C01821=1188.862,-40.963,-42.366,179.700,5.675,149.093
C01822=1188.867,-41.212,-42.354,179.698,5.675,149.094
C01823=1188.872,-41.462,-42.342,179.695,5.674,149.094
C01824=1188.878,-41.712,-42.330,179.693,5.675,149.095
C01825=1188.883,-41.961,-42.318,179.691,5.674,149.095
C01826=1188.888,-42.211,-42.306,179.688,5.673,149.096
C01827=1188.893,-42.460,-42.294,179.686,5.673,149.097
C01828=1188.898,-42.710,-42.282,179.683,5.673,149.097
C01829=1188.903,-42.960,-42.270,179.681,5.673,149.098
C01830=1188.909,-43.209,-42.258,179.679,5.672,149.099
C01831=1188.914,-43.459,-42.246,179.676,5.672,149.099
C01832=1188.919,-43.709,-42.234,179.674,5.672,149.100
C01833=1188.924,-43.959,-42.223,179.672,5.671,149.101
C01834=1188.929,-44.208,-42.210,179.669,5.671,149.101
C01835=1188.935,-44.458,-42.198,179.667,5.671,149.102
C01836=1188.939,-44.708,-42.187,179.664,5.671,149.103
C01837=1188.944,-44.957,-42.174,179.662,5.670,149.103
C01838=1188.950,-45.207,-42.162,179.659,5.669,149.104
C01839=1188.955,-45.457,-42.150,179.657,5.670,149.105
C01840=1188.961,-45.706,-42.139,179.655,5.669,149.105
C01841=1188.966,-45.955,-42.127,179.653,5.668,149.106
C01842=1188.971,-46.205,-42.115,179.650,5.668,149.106
C01843=1188.977,-46.455,-42.103,179.648,5.668,149.107
C01844=1188.981,-46.705,-42.092,179.646,5.668,149.108
C01845=1188.986,-46.954,-42.079,179.643,5.667,149.108
C01846=1188.992,-47.204,-42.067,179.640,5.667,149.109
C01847=1188.997,-47.454,-42.056,179.638,5.667,149.110
C01848=1189.002,-47.704,-42.044,179.636,5.666,149.110
C01849=1189.007,-47.954,-42.032,179.633,5.666,149.111
C01850=1189.012,-48.203,-42.020,179.631,5.666,149.112
C01851=1189.017,-48.452,-42.008,179.629,5.666,149.112
C01852=1189.023,-48.702,-41.996,179.626,5.665,149.113
C01853=1189.027,-48.952,-41.985,179.624,5.664,149.113
C01854=1189.033,-49.222,-41.973,179.621,5.664,149.114
C01855=1189.039,-49.492,-41.960,179.619,5.664,149.115
C01856=1189.045,-49.762,-41.948,179.616,5.664,149.116
C01857=1189.051,-50.033,-41.934,179.614,5.664,149.116
C01858=1189.055,-50.283,-41.923,179.611,5.663,149.117
C01859=1189.061,-50.533,-41.911,179.609,5.662,149.117
C01860=1189.065,-50.782,-41.899,179.607,5.663,149.118
C01861=1189.071,-51.031,-41.887,179.604,5.662,149.119
C01862=1189.077,-51.281,-41.876,179.601,5.662,149.120
C01863=1189.081,-51.530,-41.864,179.600,5.662,149.120
C01864=1189.087,-51.780,-41.852,179.597,5.661,149.121
C01865=1189.092,-52.030,-41.841,179.595,5.661,149.121
C01866=1189.097,-52.280,-41.829,179.592,5.661,149.122
C01867=1189.102,-52.530,-41.817,179.590,5.660,149.123
C01868=1189.107,-52.779,-41.806,179.588,5.660,149.123
C01869=1189.113,-53.029,-41.795,179.585,5.660,149.124
C01870=1189.118,-53.278,-41.783,179.583,5.660,149.125
C01871=1189.123,-53.528,-41.771,179.581,5.659,149.125
C01872=1189.128,-53.778,-41.760,179.578,5.659,149.126
C01873=1189.133,-54.028,-41.748,179.576,5.659,149.127
C01874=1189.138,-54.277,-41.737,179.573,5.659,149.127
C01875=1189.144,-54.527,-41.725,179.571,5.658,149.128
C01876=1189.150,-54.777,-41.713,179.568,5.657,149.128
C01877=1189.154,-55.026,-41.702,179.566,5.658,149.129
C01878=1189.160,-55.276,-41.690,179.564,5.657,149.130
C01879=1189.164,-55.526,-41.679,179.561,5.656,149.130
C01880=1189.170,-55.776,-41.667,179.559,5.657,149.131
C01881=1189.174,-56.025,-41.656,179.557,5.656,149.132
C01882=1189.181,-56.275,-41.644,179.555,5.656,149.132
C01883=1189.185,-56.524,-41.633,179.552,5.656,149.133
C01884=1189.191,-56.774,-41.621,179.550,5.655,149.134
C01885=1189.195,-57.024,-41.610,179.547,5.655,149.134
C01886=1189.201,-57.274,-41.598,179.546,5.655,149.135
C01887=1189.206,-57.523,-41.587,179.543,5.655,149.136
C01888=1189.211,-57.772,-41.576,179.540,5.654,149.136
C01889=1189.216,-58.023,-41.565,179.538,5.654,149.137
C01890=1189.221,-58.272,-41.553,179.536,5.654,149.137
C01891=1189.227,-58.522,-41.542,179.533,5.653,149.138
C01892=1189.232,-58.771,-41.530,179.531,5.653,149.139
C01893=1189.237,-59.021,-41.519,179.529,5.653,149.139
C01894=1189.242,-59.271,-41.507,179.526,5.652,149.140
C01895=1189.247,-59.521,-41.495,179.524,5.652,149.141
C01896=1189.253,-59.770,-41.484,179.522,5.652,149.141
C01897=1189.258,-60.020,-41.474,179.519,5.652,149.142
C01898=1189.263,-60.270,-41.462,179.517,5.651,149.143
C01899=1189.268,-60.519,-41.451,179.515,5.651,149.143
C01900=1189.274,-60.769,-41.439,179.512,5.651,149.144
C01901=1189.279,-61.018,-41.428,179.510,5.650,149.145
C01902=1189.284,-61.269,-41.417,179.508,5.651,149.145
C01903=1189.289,-61.519,-41.405,179.505,5.650,149.146
C01904=1189.294,-61.767,-41.395,179.503,5.649,149.146
C01905=1189.300,-62.017,-41.383,179.501,5.650,149.147
C01906=1189.304,-62.267,-41.371,179.498,5.649,149.148
C01907=1189.310,-62.517,-41.361,179.495,5.649,149.149
C01908=1189.315,-62.766,-41.349,179.494,5.649,149.149
C01909=1189.320,-63.016,-41.338,179.491,5.648,149.150
C01910=1189.326,-63.266,-41.326,179.489,5.648,149.150
C01911=1189.331,-63.516,-41.316,179.487,5.648,149.151
C01912=1189.336,-63.765,-41.305,179.484,5.648,149.152
C01913=1189.341,-64.015,-41.293,179.482,5.647,149.152
C01914=1189.347,-64.265,-41.283,179.480,5.648,149.153
C01915=1189.352,-64.514,-41.271,179.477,5.647,149.153
C01916=1189.357,-64.764,-41.259,179.475,5.646,149.154
C01917=1189.362,-65.013,-41.248,179.473,5.647,149.155
C01918=1189.367,-65.263,-41.238,179.470,5.646,149.155
C01919=1189.373,-65.513,-41.226,179.468,5.645,149.156
C01920=1189.378,-65.762,-41.215,179.466,5.646,149.157
C01921=1189.383,-66.013,-41.204,179.463,5.645,149.157
C01922=1189.388,-66.262,-41.193,179.461,5.645,149.158
C01923=1189.394,-66.511,-41.182,179.459,5.645,149.159
C01924=1189.399,-66.762,-41.171,179.456,5.644,149.159
C01925=1189.403,-67.011,-41.160,179.454,5.644,149.160
C01926=1189.410,-67.261,-41.149,179.452,5.644,149.161
C01927=1189.414,-67.511,-41.138,179.449,5.644,149.161
C01928=1189.419,-67.760,-41.126,179.446,5.643,149.162
C01929=1189.425,-68.010,-41.116,179.445,5.643,149.162
C01930=1189.430,-68.260,-41.104,179.442,5.643,149.163
C01931=1189.435,-68.510,-41.094,179.440,5.643,149.164
C01932=1189.440,-68.759,-41.083,179.438,5.642,149.164
C01933=1189.445,-69.009,-41.072,179.435,5.642,149.165
C01934=1189.451,-69.259,-41.060,179.433,5.642,149.166
C01935=1189.456,-69.508,-41.049,179.430,5.642,149.166
C01936=1189.461,-69.758,-41.039,179.428,5.641,149.167
C01937=1189.466,-70.007,-41.028,179.426,5.641,149.168
C01938=1189.472,-70.258,-41.017,179.424,5.641,149.168
C01939=1189.477,-70.507,-41.005,179.421,5.640,149.169
C01940=1189.482,-70.757,-40.995,179.419,5.641,149.170
C01941=1189.487,-71.007,-40.984,179.417,5.640,149.170
C01942=1189.493,-71.256,-40.974,179.414,5.639,149.171
C01943=1189.498,-71.506,-40.962,179.412,5.640,149.171
C01944=1189.503,-71.756,-40.951,179.410,5.639,149.172
C01945=1189.509,-72.005,-40.940,179.408,5.640,149.173
C01946=1189.514,-72.256,-40.930,179.405,5.639,149.173
C01947=1189.519,-72.504,-40.919,179.403,5.638,149.174
C01948=1189.525,-72.755,-40.908,179.401,5.639,149.175
C01949=1189.530,-73.004,-40.897,179.398,5.638,149.175
C01950=1189.535,-73.254,-40.886,179.396,5.638,149.176
C01951=1189.540,-73.504,-40.875,179.394,5.638,149.177
C01952=1189.545,-73.753,-40.865,179.392,5.637,149.177
C01953=1189.550,-74.003,-40.853,179.389,5.638,149.178
C01954=1189.555,-74.253,-40.843,179.387,5.637,149.179
C01955=1189.561,-74.503,-40.832,179.384,5.637,149.179
C01956=1189.566,-74.752,-40.821,179.383,5.637,149.180
C01957=1189.571,-75.002,-40.811,179.380,5.636,149.180
C01958=1189.578,-75.273,-40.799,179.377,5.636,149.181
C01959=1189.583,-75.543,-40.787,179.374,5.635,149.182
C01960=1189.588,-75.815,-40.775,179.372,5.636,149.183
C01961=1189.595,-76.085,-40.764,179.370,5.635,149.183
C01962=1189.600,-76.335,-40.753,179.368,5.635,149.184
C01963=1189.605,-76.584,-40.742,179.365,5.635,149.184
C01964=1189.610,-76.834,-40.732,179.363,5.635,149.185
C01965=1189.616,-77.084,-40.721,179.361,5.635,149.186
C01966=1189.620,-77.334,-40.710,179.359,5.634,149.186
C01967=1189.626,-77.583,-40.700,179.356,5.634,149.187
C01968=1189.631,-77.833,-40.689,179.354,5.634,149.188
C01969=1189.636,-78.082,-40.678,179.352,5.633,149.188
C01970=1189.641,-78.333,-40.668,179.349,5.633,149.189
C01971=1189.647,-78.582,-40.658,179.347,5.633,149.190
C01972=1189.652,-78.832,-40.647,179.345,5.632,149.190
C01973=1189.657,-79.081,-40.636,179.343,5.633,149.191
C01974=1189.662,-79.332,-40.625,179.340,5.632,149.192
C01975=1189.668,-79.581,-40.615,179.338,5.632,149.192
C01976=1189.673,-79.831,-40.603,179.336,5.632,149.193
C01977=1189.679,-80.081,-40.593,179.333,5.632,149.193
C01978=1189.684,-80.331,-40.583,179.331,5.632,149.194
C01979=1189.689,-80.580,-40.572,179.329,5.631,149.195
C01980=1189.694,-80.830,-40.561,179.326,5.631,149.195
C01981=1189.700,-81.080,-40.551,179.324,5.631,149.196
C01982=1189.705,-81.330,-40.540,179.322,5.630,149.197
C01983=1189.710,-81.579,-40.530,179.320,5.631,149.197
C01984=1189.715,-81.830,-40.519,179.317,5.630,149.198
C01985=1189.720,-82.079,-40.509,179.315,5.630,149.198
C01986=1189.725,-82.329,-40.498,179.313,5.630,149.199
C01987=1189.730,-82.578,-40.488,179.311,5.629,149.200
C01988=1189.736,-82.828,-40.478,179.308,5.630,149.200
C01989=1189.741,-83.078,-40.468,179.306,5.629,149.201
C01990=1189.746,-83.327,-40.457,179.304,5.628,149.202
C01991=1189.751,-83.577,-40.446,179.302,5.629,149.202
C01992=1189.757,-83.826,-40.436,179.299,5.628,149.203
C01993=1189.762,-84.077,-40.425,179.297,5.628,149.203
C01994=1189.767,-84.326,-40.415,179.295,5.628,149.204
C01995=1189.773,-84.576,-40.405,179.292,5.627,149.205
C01996=1189.778,-84.825,-40.394,179.290,5.627,149.205
C01997=1189.783,-85.075,-40.383,179.288,5.627,149.206
C01998=1189.788,-85.325,-40.373,179.286,5.627,149.207
C01999=1189.794,-85.575,-40.363,179.283,5.627,149.207
C02000=1189.799,-85.825,-40.352,179.281,5.626,149.208
C02001=1189.804,-86.074,-40.342,179.279,5.627,149.209
C02002=1189.809,-86.324,-40.332,179.276,5.626,149.209
C02003=1189.814,-86.574,-40.322,179.274,5.626,149.210
C02004=1189.820,-86.824,-40.311,179.272,5.626,149.211
C02005=1189.825,-87.073,-40.301,179.270,5.626,149.211
C02006=1189.830,-87.323,-40.291,179.267,5.625,149.212
C02007=1189.836,-87.572,-40.280,179.265,5.625,149.212
C02008=1189.841,-87.823,-40.269,179.263,5.625,149.213
C02009=1189.846,-88.072,-40.260,179.260,5.625,149.214
C02010=1189.851,-88.321,-40.249,179.258,5.625,149.214
C02011=1189.856,-88.572,-40.239,179.256,5.624,149.215
C02012=1189.862,-88.821,-40.229,179.253,5.624,149.216
C02013=1189.867,-89.071,-40.218,179.251,5.624,149.216
C02014=1189.872,-89.321,-40.208,179.249,5.623,149.217
C02015=1189.877,-89.570,-40.198,179.247,5.624,149.217
C02016=1189.883,-89.820,-40.188,179.244,5.623,149.218
C02017=1189.888,-90.070,-40.177,179.243,5.623,149.219
C02018=1189.893,-90.319,-40.167,179.240,5.623,149.219
C02019=1189.898,-90.570,-40.157,179.238,5.623,149.220
C02020=1189.903,-90.819,-40.147,179.236,5.622,149.221
C02021=1189.909,-91.068,-40.137,179.233,5.622,149.221
C02022=1189.914,-91.319,-40.126,179.232,5.622,149.222
C02023=1189.920,-91.568,-40.116,179.229,5.622,149.222
C02024=1189.925,-91.818,-40.106,179.227,5.622,149.223
C02025=1189.930,-92.068,-40.097,179.225,5.621,149.224
C02026=1189.935,-92.318,-40.086,179.222,5.621,149.224
C02027=1189.941,-92.567,-40.076,179.220,5.621,149.225
C02028=1189.946,-92.817,-40.066,179.218,5.620,149.226
C02029=1189.951,-93.067,-40.055,179.216,5.621,149.226
C02030=1189.956,-93.316,-40.046,179.213,5.620,149.227
C02031=1189.962,-93.566,-40.035,179.211,5.620,149.227
C02032=1189.967,-93.816,-40.025,179.209,5.620,149.228
C02033=1189.973,-94.066,-40.015,179.207,5.620,149.229
C02034=1189.977,-94.315,-40.005,179.204,5.620,149.229
C02035=1189.983,-94.565,-39.996,179.202,5.619,149.230
C02036=1189.988,-94.815,-39.985,179.200,5.619,149.231
C02037=1189.993,-95.065,-39.975,179.198,5.619,149.231
C02038=1189.999,-95.314,-39.965,179.195,5.619,149.232
C02039=1190.004,-95.564,-39.955,179.193,5.618,149.232
C02040=1190.009,-95.814,-39.944,179.191,5.619,149.233
C02041=1190.015,-96.064,-39.936,179.188,5.618,149.234
C02042=1190.020,-96.313,-39.925,179.187,5.618,149.234
C02043=1190.025,-96.564,-39.915,179.184,5.618,149.235
C02044=1190.030,-96.813,-39.905,179.182,5.618,149.236
C02045=1190.036,-97.062,-39.895,179.180,5.618,149.236
C02046=1190.041,-97.313,-39.885,179.177,5.617,149.237
C02047=1190.046,-97.563,-39.875,179.176,5.617,149.237
C02048=1190.051,-97.812,-39.865,179.173,5.617,149.238
C02049=1190.057,-98.062,-39.855,179.171,5.617,149.239
C02050=1190.062,-98.311,-39.845,179.169,5.616,149.239
C02051=1190.068,-98.561,-39.836,179.167,5.617,149.240
C02052=1190.073,-98.811,-39.825,179.164,5.616,149.241
C02053=1190.078,-99.060,-39.816,179.162,5.616,149.241
C02054=1190.083,-99.310,-39.806,179.160,5.616,149.242
C02055=1190.089,-99.560,-39.796,179.157,5.615,149.243
C02056=1190.093,-99.810,-39.786,179.155,5.616,149.243
C02057=1190.099,-100.060,-39.776,179.153,5.615,149.244
C02058=1190.105,-100.310,-39.766,179.151,5.615,149.244
C02059=1190.110,-100.559,-39.757,179.148,5.615,149.245
C02060=1190.115,-100.809,-39.747,179.147,5.615,149.246
C02061=1190.120,-101.059,-39.737,179.144,5.614,149.246
C02062=1190.126,-101.330,-39.726,179.142,5.615,149.247
C02063=1190.132,-101.602,-39.716,179.139,5.614,149.248
C02064=1190.137,-101.873,-39.705,179.137,5.614,149.248
C02065=1190.143,-102.146,-39.694,179.135,5.614,149.249
C02066=1190.148,-102.395,-39.684,179.132,5.614,149.250
C02067=1190.154,-102.644,-39.674,179.130,5.613,149.250
C02068=1190.159,-102.894,-39.665,179.128,5.613,149.251
C02069=1190.165,-103.144,-39.655,179.126,5.613,149.252
C02070=1190.169,-103.394,-39.645,179.124,5.613,149.252
C02071=1190.175,-103.644,-39.636,179.121,5.612,149.253
C02072=1190.180,-103.893,-39.625,179.119,5.613,149.253
C02073=1190.185,-104.143,-39.617,179.117,5.612,149.254
C02074=1190.191,-104.393,-39.606,179.115,5.613,149.255
C02075=1190.196,-104.642,-39.597,179.113,5.612,149.255
C02076=1190.202,-104.892,-39.587,179.111,5.612,149.256
C02077=1190.206,-105.142,-39.577,179.108,5.612,149.257
C02078=1190.212,-105.392,-39.568,179.106,5.612,149.257
C02079=1190.217,-105.641,-39.558,179.104,5.611,149.258
C02080=1190.222,-105.891,-39.548,179.102,5.611,149.258
C02081=1190.228,-106.141,-39.539,179.099,5.611,149.259
C02082=1190.233,-106.390,-39.529,179.097,5.611,149.260
C02083=1190.238,-106.640,-39.520,179.095,5.611,149.260
C02084=1190.243,-106.890,-39.509,179.092,5.610,149.261
C02085=1190.249,-107.140,-39.501,179.091,5.610,149.261
C02086=1190.254,-107.390,-39.490,179.088,5.610,149.262
C02087=1190.259,-107.640,-39.481,179.086,5.610,149.263
C02088=1190.265,-107.889,-39.471,179.084,5.609,149.263
C02089=1190.270,-108.139,-39.462,179.082,5.610,149.264
C02090=1190.276,-108.389,-39.452,179.080,5.609,149.265
C02091=1190.281,-108.639,-39.443,179.078,5.609,149.265
C02092=1190.286,-108.888,-39.434,179.075,5.609,149.266
C02093=1190.291,-109.139,-39.424,179.073,5.609,149.266
C02094=1190.296,-109.388,-39.414,179.071,5.609,149.267
C02095=1190.302,-109.638,-39.405,179.069,5.609,149.268
C02096=1190.307,-109.887,-39.395,179.066,5.608,149.268
C02097=1190.313,-110.137,-39.386,179.065,5.608,149.269
C02098=1190.317,-110.387,-39.376,179.062,5.608,149.270
C02099=1190.323,-110.637,-39.366,179.060,5.608,149.270
C02100=1190.328,-110.887,-39.358,179.058,5.607,149.271
C02101=1190.333,-111.136,-39.348,179.056,5.608,149.271
C02102=1190.339,-111.386,-39.338,179.053,5.607,149.272
C02103=1190.344,-111.635,-39.329,179.051,5.607,149.273
C02104=1190.350,-111.885,-39.319,179.049,5.607,149.273
C02105=1190.355,-112.135,-39.310,179.047,5.607,149.274
C02106=1190.360,-112.384,-39.301,179.044,5.607,149.275
C02107=1190.366,-112.635,-39.291,179.043,5.607,149.275
C02108=1190.371,-112.884,-39.282,179.040,5.606,149.276
C02109=1190.376,-113.135,-39.272,179.039,5.606,149.276
C02110=1190.381,-113.385,-39.263,179.036,5.606,149.277
C02111=1190.386,-113.634,-39.253,179.034,5.606,149.277
C02112=1190.392,-113.884,-39.244,179.032,5.606,149.278
C02113=1190.397,-114.134,-39.235,179.029,5.606,149.279
C02114=1190.402,-114.383,-39.225,179.027,5.605,149.279
C02115=1190.408,-114.633,-39.216,179.025,5.606,149.280
C02116=1190.413,-114.883,-39.207,179.023,5.605,149.281
C02117=1190.418,-115.132,-39.197,179.021,5.605,149.281
C02118=1190.424,-115.383,-39.188,179.019,5.604,149.282
C02119=1190.429,-115.632,-39.179,179.017,5.605,149.282
C02120=1190.434,-115.882,-39.169,179.014,5.604,149.283
C02121=1190.440,-116.132,-39.160,179.012,5.604,149.284
C02122=1190.445,-116.382,-39.151,179.010,5.604,149.284
C02123=1190.450,-116.631,-39.142,179.008,5.604,149.285
C02124=1190.456,-116.881,-39.132,179.005,5.604,149.286
C02125=1190.461,-117.131,-39.123,179.004,5.604,149.286
C02126=1190.466,-117.381,-39.114,179.001,5.603,149.287
C02127=1190.472,-117.631,-39.104,179.000,5.603,149.287
C02128=1190.477,-117.880,-39.095,178.997,5.603,149.288
C02129=1190.482,-118.130,-39.086,178.995,5.603,149.288
C02130=1190.487,-118.380,-39.077,178.993,5.603,149.289
C02131=1190.493,-118.630,-39.068,178.991,5.603,149.290
C02132=1190.498,-118.879,-39.058,178.988,5.602,149.290
C02133=1190.503,-119.129,-39.049,178.986,5.603,149.291
C02134=1190.509,-119.378,-39.041,178.984,5.602,149.292
C02135=1190.515,-119.628,-39.031,178.982,5.602,149.292
C02136=1190.520,-119.878,-39.021,178.980,5.601,149.293
C02137=1190.525,-120.127,-39.013,178.978,5.602,149.294
C02138=1190.530,-120.377,-39.004,178.975,5.601,149.294
C02139=1190.536,-120.627,-38.994,178.973,5.602,149.295
C02140=1190.541,-120.877,-38.985,178.971,5.601,149.295
C02141=1190.546,-121.127,-38.976,178.969,5.601,149.296
C02142=1190.551,-121.376,-38.967,178.967,5.600,149.296
C02143=1190.556,-121.626,-38.958,178.965,5.601,149.297
C02144=1190.562,-121.876,-38.948,178.963,5.600,149.298
C02145=1190.567,-122.126,-38.939,178.961,5.600,149.298
C02146=1190.572,-122.376,-38.931,178.958,5.600,149.299
C02147=1190.578,-122.626,-38.922,178.956,5.600,149.300
C02148=1190.583,-122.876,-38.913,178.954,5.599,149.300
C02149=1190.589,-123.126,-38.903,178.952,5.600,149.301
C02150=1190.594,-123.374,-38.894,178.950,5.600,149.301
C02151=1190.599,-123.624,-38.885,178.948,5.599,149.302
C02152=1190.604,-123.874,-38.876,178.946,5.600,149.303
C02153=1190.610,-124.124,-38.867,178.943,5.599,149.303
C02154=1190.615,-124.374,-38.858,178.941,5.599,149.304
C02155=1190.621,-124.624,-38.849,178.939,5.599,149.304
C02156=1190.626,-124.874,-38.840,178.937,5.599,149.305
C02157=1190.631,-125.124,-38.831,178.935,5.598,149.306
C02158=1190.636,-125.374,-38.822,178.933,5.599,149.306
C02159=1190.641,-125.623,-38.813,178.931,5.598,149.307
C02160=1190.647,-125.873,-38.805,178.929,5.598,149.307
C02161=1190.653,-126.123,-38.795,178.926,5.597,149.308
C02162=1190.658,-126.373,-38.786,178.924,5.598,149.309
C02163=1190.663,-126.622,-38.778,178.922,5.597,149.309
C02164=1190.669,-126.872,-38.769,178.920,5.598,149.310
C02165=1190.674,-127.122,-38.760,178.918,5.597,149.310
C02166=1190.252,-127.133,-38.798,178.914,5.601,149.312
C02167=1190.247,-126.883,-38.807,178.916,5.601,149.312
C02168=1190.241,-126.633,-38.817,178.919,5.601,149.311
C02169=1190.236,-126.383,-38.826,178.920,5.601,149.311
C02170=1190.231,-126.133,-38.835,178.922,5.601,149.310
C02171=1190.226,-125.884,-38.844,178.925,5.601,149.309
C02172=1190.221,-125.634,-38.852,178.927,5.601,149.309
C02173=1190.216,-125.384,-38.861,178.929,5.602,149.308
C02174=1190.210,-125.135,-38.870,178.931,5.601,149.307
C02175=1190.204,-124.885,-38.879,178.933,5.602,149.307
C02176=1190.199,-124.635,-38.888,178.935,5.602,149.306
C02177=1190.194,-124.385,-38.897,178.937,5.603,149.306
C02178=1190.188,-124.135,-38.906,178.940,5.602,149.305
C02179=1190.183,-123.885,-38.915,178.942,5.603,149.305
C02180=1190.178,-123.636,-38.925,178.944,5.603,149.304
C02181=1190.173,-123.386,-38.933,178.946,5.603,149.303
C02182=1190.167,-123.136,-38.943,178.948,5.603,149.303
C02183=1190.161,-122.887,-38.952,178.950,5.604,149.302
C02184=1190.156,-122.637,-38.960,178.952,5.603,149.301
C02185=1190.151,-122.387,-38.969,178.955,5.604,149.301
C02186=1190.146,-122.137,-38.978,178.957,5.604,149.300
C02187=1190.140,-121.887,-38.988,178.959,5.604,149.300
C02188=1190.135,-121.637,-38.997,178.961,5.604,149.299
C02189=1190.130,-121.388,-39.006,178.963,5.605,149.298
C02190=1190.125,-121.138,-39.015,178.965,5.604,149.298
C02191=1190.120,-120.888,-39.024,178.967,5.604,149.297
C02192=1190.114,-120.638,-39.034,178.969,5.605,149.297
C02193=1190.109,-120.388,-39.042,178.972,5.604,149.296
C02194=1190.103,-120.138,-39.051,178.974,5.605,149.295
C02195=1190.099,-119.889,-39.061,178.976,5.605,149.295
C02196=1190.093,-119.639,-39.070,178.978,5.605,149.294
C02197=1190.088,-119.389,-39.079,178.980,5.605,149.293
C02198=1190.082,-119.139,-39.088,178.982,5.606,149.293
C02199=1190.077,-118.889,-39.097,178.984,5.605,149.292
C02200=1190.071,-118.641,-39.107,178.987,5.606,149.292
C02201=1190.066,-118.391,-39.116,178.989,5.606,149.291
C02202=1190.061,-118.141,-39.125,178.991,5.607,149.291
C02203=1190.056,-117.891,-39.134,178.993,5.606,149.290
C02204=1190.050,-117.642,-39.144,178.995,5.607,149.289
C02205=1190.045,-117.392,-39.153,178.997,5.607,149.289
C02206=1190.040,-117.142,-39.162,179.000,5.607,149.288
C02207=1190.034,-116.892,-39.171,179.002,5.607,149.287
C02208=1190.029,-116.642,-39.181,179.004,5.607,149.287
C02209=1190.024,-116.393,-39.190,179.006,5.607,149.286
C02210=1190.019,-116.143,-39.199,179.008,5.608,149.286
C02211=1190.013,-115.893,-39.208,179.010,5.608,149.285
C02212=1190.008,-115.643,-39.218,179.013,5.608,149.284
C02213=1190.003,-115.393,-39.227,179.014,5.608,149.284
C02214=1189.997,-115.143,-39.236,179.017,5.608,149.283
C02215=1189.992,-114.894,-39.246,179.019,5.608,149.283
C02216=1189.987,-114.644,-39.255,179.021,5.609,149.282
C02217=1189.981,-114.394,-39.264,179.023,5.608,149.281
C02218=1189.976,-114.145,-39.274,179.026,5.609,149.281
C02219=1189.970,-113.895,-39.283,179.028,5.609,149.280
C02220=1189.965,-113.645,-39.292,179.030,5.610,149.280
C02221=1189.960,-113.396,-39.302,179.032,5.609,149.279
C02222=1189.954,-113.145,-39.311,179.034,5.610,149.278
C02223=1189.949,-112.895,-39.320,179.036,5.610,149.278
C02224=1189.945,-112.646,-39.330,179.038,5.610,149.277
C02225=1189.939,-112.395,-39.340,179.040,5.610,149.276
C02226=1189.934,-112.146,-39.349,179.043,5.610,149.276
C02227=1189.928,-111.896,-39.359,179.045,5.610,149.275
C02228=1189.923,-111.646,-39.368,179.047,5.611,149.275
C02229=1189.918,-111.397,-39.377,179.049,5.611,149.274
C02230=1189.912,-111.147,-39.387,179.052,5.611,149.273
C02231=1189.907,-110.898,-39.396,179.053,5.611,149.273
C02232=1189.901,-110.647,-39.406,179.056,5.611,149.272
C02233=1189.896,-110.398,-39.415,179.058,5.611,149.271
C02234=1189.891,-110.148,-39.424,179.060,5.612,149.271
C02235=1189.885,-109.898,-39.434,179.062,5.611,149.270
C02236=1189.880,-109.649,-39.443,179.065,5.612,149.270
C02237=1189.875,-109.399,-39.453,179.067,5.612,149.269
C02238=1189.870,-109.150,-39.462,179.069,5.613,149.269
C02239=1189.864,-108.899,-39.472,179.071,5.612,149.268
C02240=1189.860,-108.649,-39.482,179.074,5.613,149.267
C02241=1189.854,-108.400,-39.491,179.076,5.613,149.267
C02242=1189.849,-108.150,-39.501,179.078,5.613,149.266
C02243=1189.844,-107.900,-39.510,179.080,5.614,149.265
C02244=1189.838,-107.651,-39.520,179.082,5.613,149.265
C02245=1189.833,-107.401,-39.529,179.085,5.614,149.264
C02246=1189.827,-107.151,-39.539,179.086,5.614,149.263
C02247=1189.822,-106.901,-39.548,179.089,5.614,149.263
C02248=1189.817,-106.651,-39.559,179.091,5.614,149.262
C02249=1189.812,-106.401,-39.568,179.093,5.615,149.262
C02250=1189.806,-106.152,-39.578,179.095,5.615,149.261
C02251=1189.801,-105.902,-39.587,179.098,5.615,149.260
C02252=1189.796,-105.652,-39.597,179.100,5.615,149.260
C02253=1189.790,-105.403,-39.606,179.102,5.615,149.259
C02254=1189.785,-105.153,-39.616,179.104,5.615,149.258
C02255=1189.780,-104.904,-39.626,179.106,5.616,149.258
C02256=1189.775,-104.653,-39.636,179.108,5.615,149.257
C02257=1189.770,-104.404,-39.645,179.111,5.616,149.257
C02258=1189.764,-104.154,-39.655,179.113,5.616,149.256
C02259=1189.759,-103.904,-39.664,179.115,5.616,149.255
C02260=1189.753,-103.655,-39.674,179.117,5.616,149.255
C02261=1189.747,-103.405,-39.684,179.120,5.616,149.254
C02262=1189.743,-103.155,-39.694,179.122,5.617,149.253
C02263=1189.737,-102.904,-39.703,179.124,5.617,149.253
C02264=1189.732,-102.655,-39.713,179.126,5.617,149.252
C02265=1189.727,-102.406,-39.723,179.128,5.617,149.252
C02266=1189.722,-102.156,-39.732,179.131,5.618,149.251
C02267=1189.716,-101.884,-39.744,179.133,5.617,149.250
C02268=1189.710,-101.612,-39.754,179.136,5.618,149.250
C02269=1189.705,-101.341,-39.765,179.138,5.618,149.249
C02270=1189.698,-101.070,-39.775,179.140,5.618,149.248
C02271=1189.693,-100.820,-39.785,179.142,5.618,149.248
C02272=1189.688,-100.570,-39.795,179.145,5.618,149.247
C02273=1189.683,-100.320,-39.804,179.147,5.619,149.247
C02274=1189.678,-100.071,-39.815,179.149,5.619,149.246
C02275=1189.672,-99.821,-39.825,179.151,5.619,149.245
C02276=1189.667,-99.571,-39.834,179.154,5.620,149.245
C02277=1189.662,-99.321,-39.844,179.156,5.619,149.244
C02278=1189.657,-99.072,-39.854,179.158,5.620,149.243
C02279=1189.651,-98.822,-39.864,179.160,5.620,149.243
C02280=1189.646,-98.572,-39.874,179.162,5.620,149.242
C02281=1189.641,-98.322,-39.884,179.164,5.620,149.241
C02282=1189.636,-98.073,-39.894,179.167,5.620,149.241
C02283=1189.630,-97.823,-39.904,179.169,5.620,149.240
C02284=1189.625,-97.573,-39.913,179.171,5.621,149.240
C02285=1189.620,-97.323,-39.923,179.174,5.621,149.239
C02286=1189.614,-97.073,-39.934,179.176,5.621,149.238
C02287=1189.609,-96.824,-39.943,179.178,5.622,149.238
C02288=1189.604,-96.575,-39.953,179.180,5.622,149.237
C02289=1189.599,-96.324,-39.963,179.182,5.622,149.236
C02290=1189.593,-96.074,-39.974,179.185,5.622,149.236
C02291=1189.588,-95.825,-39.983,179.187,5.622,149.235
C02292=1189.582,-95.575,-39.993,179.189,5.622,149.235
C02293=1189.577,-95.325,-40.004,179.192,5.622,149.234
C02294=1189.572,-95.075,-40.013,179.194,5.623,149.233
C02295=1189.567,-94.826,-40.023,179.196,5.623,149.233
C02296=1189.561,-94.576,-40.033,179.198,5.624,149.232
C02297=1189.556,-94.326,-40.044,179.200,5.623,149.231
C02298=1189.551,-94.077,-40.053,179.203,5.624,149.231
C02299=1189.546,-93.827,-40.064,179.204,5.624,149.230
C02300=1189.540,-93.578,-40.074,179.207,5.624,149.230
C02301=1189.535,-93.327,-40.084,179.209,5.624,149.229
C02302=1189.530,-93.078,-40.093,179.211,5.624,149.228
C02303=1189.524,-92.828,-40.104,179.214,5.625,149.228
C02304=1189.519,-92.578,-40.114,179.216,5.624,149.227
C02305=1189.514,-92.328,-40.124,179.218,5.625,149.226
C02306=1189.509,-92.079,-40.134,179.220,5.625,149.226
C02307=1189.504,-91.829,-40.145,179.223,5.625,149.225
C02308=1189.498,-91.579,-40.155,179.225,5.625,149.225
C02309=1189.493,-91.330,-40.165,179.227,5.626,149.224
C02310=1189.488,-91.080,-40.175,179.229,5.626,149.223
C02311=1189.483,-90.830,-40.185,179.232,5.626,149.223
C02312=1189.477,-90.581,-40.195,179.234,5.626,149.222
C02313=1189.472,-90.330,-40.206,179.236,5.626,149.221
C02314=1189.467,-90.081,-40.216,179.238,5.627,149.221
C02315=1189.461,-89.831,-40.226,179.241,5.626,149.220
C02316=1189.457,-89.581,-40.236,179.243,5.627,149.220
C02317=1189.451,-89.332,-40.247,179.245,5.628,149.219
C02318=1189.446,-89.082,-40.257,179.247,5.627,149.218
C02319=1189.441,-88.832,-40.267,179.250,5.628,149.218
C02320=1189.435,-88.583,-40.278,179.252,5.628,149.217
C02321=1189.429,-88.333,-40.288,179.254,5.628,149.216
C02322=1189.425,-88.083,-40.298,179.256,5.628,149.216
C02323=1189.419,-87.834,-40.308,179.259,5.629,149.215
C02324=1189.414,-87.584,-40.318,179.261,5.629,149.214
C02325=1189.409,-87.334,-40.329,179.263,5.629,149.214
C02326=1189.403,-87.084,-40.339,179.266,5.629,149.213
C02327=1189.398,-86.834,-40.349,179.268,5.629,149.212
C02328=1189.393,-86.584,-40.360,179.270,5.630,149.212
C02329=1189.388,-86.335,-40.369,179.273,5.630,149.211
C02330=1189.383,-86.085,-40.380,179.274,5.630,149.211
C02331=1189.377,-85.835,-40.390,179.277,5.631,149.210
C02332=1189.372,-85.585,-40.401,179.279,5.630,149.209
C02333=1189.367,-85.336,-40.412,179.281,5.631,149.209
C02334=1189.361,-85.087,-40.422,179.283,5.631,149.208
C02335=1189.356,-84.836,-40.432,179.286,5.631,149.207
C02336=1189.351,-84.587,-40.443,179.288,5.632,149.207
C02337=1189.346,-84.337,-40.453,179.290,5.631,149.206
C02338=1189.340,-84.087,-40.463,179.293,5.632,149.206
C02339=1189.336,-83.837,-40.473,179.294,5.632,149.205
C02340=1189.330,-83.588,-40.484,179.297,5.632,149.204
C02341=1189.325,-83.339,-40.494,179.300,5.633,149.204
C02342=1189.320,-83.088,-40.505,179.301,5.633,149.203
C02343=1189.314,-82.839,-40.515,179.304,5.633,149.202
C02344=1189.309,-82.589,-40.526,179.306,5.633,149.202
C02345=1189.304,-82.339,-40.536,179.308,5.633,149.201
C02346=1189.299,-82.089,-40.547,179.311,5.634,149.201
C02347=1189.294,-81.840,-40.558,179.313,5.634,149.200
C02348=1189.288,-81.590,-40.568,179.315,5.634,149.199
C02349=1189.283,-81.340,-40.578,179.317,5.634,149.199
C02350=1189.277,-81.091,-40.589,179.320,5.634,149.198
C02351=1189.273,-80.841,-40.600,179.323,5.635,149.197
C02352=1189.267,-80.591,-40.610,179.324,5.635,149.197
C02353=1189.262,-80.341,-40.621,179.327,5.635,149.196
C02354=1189.256,-80.092,-40.631,179.329,5.635,149.195
C02355=1189.252,-79.842,-40.642,179.331,5.636,149.195
C02356=1189.246,-79.592,-40.652,179.334,5.636,149.194
C02357=1189.241,-79.342,-40.663,179.336,5.636,149.193
C02358=1189.236,-79.093,-40.673,179.338,5.636,149.193
C02359=1189.231,-78.843,-40.684,179.340,5.636,149.192
C02360=1189.225,-78.594,-40.695,179.343,5.636,149.192
C02361=1189.220,-78.343,-40.705,179.345,5.637,149.191
C02362=1189.215,-78.094,-40.716,179.347,5.637,149.190
C02363=1189.210,-77.844,-40.727,179.350,5.637,149.190
C02364=1189.204,-77.595,-40.737,179.352,5.638,149.189
C02365=1189.199,-77.345,-40.749,179.354,5.638,149.188
C02366=1189.193,-77.095,-40.759,179.357,5.638,149.188
C02367=1189.188,-76.845,-40.770,179.358,5.638,149.187
C02368=1189.183,-76.596,-40.780,179.361,5.639,149.187
C02369=1189.178,-76.346,-40.791,179.364,5.639,149.186
C02370=1189.172,-76.096,-40.801,179.365,5.639,149.185
C02371=1189.167,-75.825,-40.813,179.368,5.639,149.185
C02372=1189.161,-75.555,-40.825,179.371,5.640,149.184
C02373=1189.155,-75.284,-40.836,179.373,5.640,149.183
C02374=1189.150,-75.013,-40.849,179.375,5.640,149.183
C02375=1189.144,-74.763,-40.859,179.378,5.640,149.182
C02376=1189.140,-74.513,-40.870,179.380,5.641,149.181
C02377=1189.134,-74.264,-40.880,179.382,5.641,149.181
C02378=1189.129,-74.014,-40.891,179.385,5.641,149.180
C02379=1189.124,-73.765,-40.902,179.387,5.641,149.179
C02380=1189.119,-73.514,-40.912,179.389,5.642,149.179
C02381=1189.113,-73.265,-40.924,179.392,5.642,149.178
C02382=1189.108,-73.015,-40.934,179.394,5.642,149.177
C02383=1189.103,-72.765,-40.946,179.396,5.642,149.177
C02384=1189.097,-72.516,-40.956,179.399,5.643,149.176
C02385=1189.093,-72.266,-40.967,179.401,5.642,149.175
C02386=1189.087,-72.017,-40.977,179.403,5.643,149.175
C02387=1189.081,-71.766,-40.989,179.405,5.643,149.174
C02388=1189.077,-71.516,-41.000,179.408,5.643,149.174
C02389=1189.071,-71.267,-41.010,179.411,5.644,149.173
C02390=1189.066,-71.017,-41.021,179.412,5.644,149.172
C02391=1189.061,-70.768,-41.032,179.415,5.644,149.172
C02392=1189.055,-70.518,-41.043,179.418,5.645,149.171
C02393=1189.051,-70.268,-41.055,179.419,5.645,149.170
C02394=1189.045,-70.019,-41.065,179.422,5.645,149.170
C02395=1189.040,-69.769,-41.076,179.424,5.645,149.169
C02396=1189.034,-69.519,-41.087,179.426,5.645,149.169
C02397=1189.029,-69.270,-41.098,179.429,5.646,149.168
C02398=1189.024,-69.019,-41.109,179.431,5.646,149.167
C02399=1189.019,-68.770,-41.120,179.433,5.646,149.166
C02400=1189.013,-68.520,-41.131,179.436,5.647,149.166
C02401=1189.008,-68.271,-41.142,179.438,5.646,149.165
C02402=1189.003,-68.021,-41.153,179.440,5.647,149.165
C02403=1188.998,-67.771,-41.164,179.443,5.648,149.164
C02404=1188.992,-67.522,-41.175,179.445,5.647,149.163
C02405=1188.987,-67.272,-41.186,179.447,5.648,149.163
C02406=1188.983,-67.022,-41.197,179.450,5.648,149.162
C02407=1188.977,-66.773,-41.208,179.452,5.648,149.161
C02408=1188.972,-66.522,-41.219,179.454,5.648,149.161
C02409=1188.967,-66.273,-41.231,179.457,5.649,149.160
C02410=1188.962,-66.024,-41.242,179.459,5.649,149.160
C02411=1188.956,-65.773,-41.253,179.461,5.649,149.159
C02412=1188.951,-65.524,-41.264,179.464,5.650,149.158
C02413=1188.946,-65.275,-41.275,179.465,5.650,149.158
C02414=1188.941,-65.025,-41.285,179.468,5.650,149.157
C02415=1188.935,-64.775,-41.297,179.471,5.651,149.156
C02416=1188.930,-64.526,-41.308,179.473,5.650,149.156
C02417=1188.925,-64.275,-41.319,179.475,5.651,149.155
C02418=1188.920,-64.026,-41.331,179.478,5.651,149.154
C02419=1188.914,-63.777,-41.342,179.480,5.651,149.154
C02420=1188.909,-63.526,-41.352,179.482,5.652,149.153
C02421=1188.904,-63.276,-41.364,179.485,5.652,149.152
C02422=1188.899,-63.027,-41.375,179.487,5.652,149.152
C02423=1188.893,-62.778,-41.387,179.489,5.652,149.151
C02424=1188.888,-62.527,-41.398,179.492,5.653,149.151
C02425=1188.884,-62.278,-41.409,179.494,5.653,149.150
C02426=1188.878,-62.028,-41.420,179.496,5.653,149.149
C02427=1188.873,-61.779,-41.432,179.499,5.654,149.149
C02428=1188.868,-61.529,-41.442,179.501,5.654,149.148
C02429=1188.862,-61.279,-41.454,179.503,5.654,149.147
C02430=1188.857,-61.030,-41.465,179.506,5.655,149.147
C02431=1188.852,-60.780,-41.477,179.508,5.655,149.146
C02432=1188.847,-60.530,-41.488,179.510,5.655,149.145
C02433=1188.842,-60.281,-41.499,179.513,5.655,149.145
C02434=1188.836,-60.031,-41.510,179.515,5.655,149.144
C02435=1188.831,-59.781,-41.522,179.517,5.656,149.144
C02436=1188.826,-59.531,-41.533,179.520,5.656,149.143
C02437=1188.821,-59.281,-41.545,179.522,5.656,149.142
C02438=1188.815,-59.032,-41.556,179.524,5.657,149.142
C02439=1188.810,-58.783,-41.568,179.527,5.657,149.141
C02440=1188.805,-58.532,-41.578,179.529,5.657,149.140
C02441=1188.800,-58.282,-41.590,179.532,5.657,149.140
C02442=1188.795,-58.034,-41.601,179.534,5.658,149.139
C02443=1188.789,-57.784,-41.613,179.536,5.658,149.138
C02444=1188.785,-57.534,-41.624,179.538,5.658,149.138
C02445=1188.779,-57.284,-41.636,179.541,5.659,149.137
C02446=1188.774,-57.034,-41.647,179.543,5.659,149.136
C02447=1188.768,-56.785,-41.659,179.545,5.659,149.136
C02448=1188.764,-56.536,-41.670,179.548,5.659,149.135
C02449=1188.758,-56.286,-41.682,179.550,5.660,149.135
C02450=1188.753,-56.035,-41.693,179.552,5.660,149.134
C02451=1188.748,-55.785,-41.704,179.555,5.660,149.133
C02452=1188.743,-55.536,-41.715,179.558,5.661,149.132
C02453=1188.737,-55.287,-41.727,179.559,5.661,149.132
C02454=1188.732,-55.037,-41.739,179.562,5.661,149.131
C02455=1188.727,-54.787,-41.750,179.565,5.662,149.131
C02456=1188.722,-54.537,-41.762,179.567,5.662,149.130
C02457=1188.717,-54.287,-41.774,179.569,5.662,149.129
C02458=1188.712,-54.038,-41.785,179.572,5.662,149.129
C02459=1188.706,-53.789,-41.796,179.574,5.663,149.128
C02460=1188.702,-53.539,-41.808,179.576,5.663,149.128
C02461=1188.696,-53.289,-41.820,179.578,5.663,149.127
C02462=1188.691,-53.039,-41.831,179.581,5.664,149.126
C02463=1188.686,-52.789,-41.843,179.583,5.663,149.125
C02464=1188.681,-52.539,-41.855,179.585,5.664,149.125
C02465=1188.675,-52.291,-41.866,179.588,5.665,149.124
C02466=1188.670,-52.041,-41.878,179.591,5.665,149.124
C02467=1188.665,-51.792,-41.889,179.593,5.665,149.123
C02468=1188.660,-51.542,-41.901,179.595,5.666,149.122
C02469=1188.655,-51.292,-41.913,179.598,5.666,149.122
C02470=1188.650,-51.042,-41.925,179.600,5.666,149.121
C02471=1188.644,-50.792,-41.936,179.602,5.666,149.120
C02472=1188.639,-50.543,-41.947,179.605,5.667,149.120
C02473=1188.634,-50.293,-41.959,179.607,5.667,149.119
C02474=1188.628,-50.043,-41.971,179.609,5.667,149.118
C02475=1188.623,-49.773,-41.984,179.612,5.667,149.118
C02476=1188.618,-49.503,-41.997,179.615,5.668,149.117
C02477=1188.612,-49.233,-42.010,179.617,5.668,149.116
C02478=1188.606,-48.962,-42.022,179.620,5.669,149.116
C02479=1188.602,-48.713,-42.034,179.622,5.669,149.115
C02480=1188.596,-48.463,-42.046,179.624,5.669,149.114
C02481=1188.590,-48.214,-42.057,179.627,5.670,149.114
C02482=1188.586,-47.964,-42.069,179.630,5.670,149.113
C02483=1188.580,-47.714,-42.080,179.631,5.670,149.112
C02484=1188.575,-47.464,-42.092,179.634,5.671,149.112
C02485=1188.570,-47.215,-42.104,179.636,5.671,149.111
C02486=1188.565,-46.965,-42.116,179.639,5.672,149.111
C02487=1188.560,-46.716,-42.128,179.641,5.671,149.110
C02488=1188.554,-46.466,-42.140,179.643,5.672,149.109
C02489=1188.549,-46.216,-42.151,179.646,5.672,149.108
C02490=1188.544,-45.967,-42.164,179.648,5.673,149.108
C02491=1188.539,-45.717,-42.176,179.650,5.673,149.107
C02492=1188.534,-45.467,-42.187,179.653,5.673,149.107
C02493=1188.529,-45.217,-42.199,179.656,5.674,149.106
C02494=1188.524,-44.968,-42.212,179.657,5.674,149.105
C02495=1188.518,-44.718,-42.223,179.660,5.674,149.105
C02496=1188.513,-44.468,-42.235,179.663,5.675,149.104
C02497=1188.508,-44.219,-42.247,179.665,5.675,149.103
C02498=1188.503,-43.969,-42.259,179.667,5.675,149.103
C02499=1188.497,-43.720,-42.271,179.669,5.675,149.102
C02500=1188.492,-43.470,-42.282,179.672,5.676,149.101
C02501=1188.487,-43.221,-42.295,179.675,5.676,149.101
C02502=1188.482,-42.971,-42.307,179.676,5.676,149.100
C02503=1188.476,-42.721,-42.318,179.679,5.677,149.100
C02504=1188.471,-42.472,-42.331,179.682,5.677,149.099
C02505=1188.466,-42.222,-42.342,179.684,5.678,149.098
C02506=1188.461,-41.972,-42.354,179.686,5.678,149.098
C02507=1188.456,-41.723,-42.367,179.689,5.678,149.097
C02508=1188.450,-41.473,-42.379,179.691,5.679,149.096
C02509=1188.445,-41.223,-42.391,179.694,5.679,149.096
C02510=1188.441,-40.974,-42.403,179.696,5.679,149.095
C02511=1188.436,-40.723,-42.415,179.698,5.680,149.094
C02512=1188.431,-40.474,-42.427,179.701,5.680,149.094
C02513=1188.425,-40.224,-42.439,179.704,5.680,149.093
C02514=1188.420,-39.975,-42.452,179.705,5.680,149.093
C02515=1188.415,-39.725,-42.464,179.708,5.681,149.092
C02516=1188.410,-39.475,-42.475,179.710,5.681,149.091
C02517=1188.405,-39.226,-42.488,179.713,5.682,149.090
C02518=1188.399,-38.976,-42.500,179.715,5.683,149.090
C02519=1188.394,-38.727,-42.512,179.717,5.682,149.089
C02520=1188.389,-38.477,-42.524,179.720,5.683,149.089
C02521=1188.384,-38.227,-42.537,179.723,5.683,149.088
C02522=1188.378,-37.977,-42.549,179.725,5.684,149.087
C02523=1188.373,-37.728,-42.561,179.727,5.684,149.087
C02524=1188.368,-37.478,-42.573,179.730,5.684,149.086
C02525=1188.363,-37.229,-42.585,179.732,5.685,149.085
C02526=1188.358,-36.979,-42.597,179.735,5.685,149.085
C02527=1188.353,-36.730,-42.610,179.737,5.685,149.084
C02528=1188.347,-36.480,-42.621,179.739,5.685,149.083
C02529=1188.342,-36.231,-42.634,179.742,5.686,149.083
C02530=1188.337,-35.981,-42.646,179.744,5.687,149.082
C02531=1188.332,-35.731,-42.659,179.747,5.687,149.082
C02532=1188.327,-35.481,-42.671,179.749,5.687,149.081
C02533=1188.322,-35.231,-42.683,179.751,5.687,149.080
C02534=1188.316,-34.981,-42.695,179.754,5.688,149.080
C02535=1188.311,-34.732,-42.708,179.756,5.689,149.079
C02536=1188.306,-34.483,-42.720,179.758,5.688,149.078
C02537=1188.301,-34.233,-42.732,179.761,5.689,149.078
C02538=1188.296,-33.984,-42.745,179.763,5.689,149.077
C02539=1188.290,-33.734,-42.757,179.766,5.690,149.076
C02540=1188.286,-33.484,-42.770,179.769,5.690,149.076
C02541=1188.280,-33.234,-42.782,179.771,5.690,149.075
C02542=1188.275,-32.984,-42.794,179.773,5.691,149.075
C02543=1188.270,-32.735,-42.807,179.775,5.691,149.074
C02544=1188.264,-32.485,-42.819,179.778,5.692,149.073
C02545=1188.259,-32.236,-42.831,179.781,5.692,149.072
C02546=1188.254,-31.986,-42.844,179.782,5.692,149.072
C02547=1188.249,-31.736,-42.856,179.785,5.693,149.071
C02548=1188.244,-31.486,-42.869,179.788,5.693,149.071
C02549=1188.239,-31.237,-42.881,179.790,5.694,149.070
C02550=1188.234,-30.987,-42.893,179.793,5.694,149.069
C02551=1188.229,-30.738,-42.906,179.795,5.694,149.069
C02552=1188.223,-30.489,-42.918,179.797,5.695,149.068
C02553=1188.219,-30.239,-42.931,179.800,5.695,149.067
C02554=1188.214,-29.989,-42.943,179.802,5.696,149.067
C02555=1188.208,-29.739,-42.956,179.805,5.696,149.066
C02556=1188.203,-29.490,-42.969,179.807,5.696,149.065
C02557=1188.198,-29.241,-42.981,179.810,5.696,149.065
C02558=1188.193,-28.991,-42.993,179.812,5.697,149.064
C02559=1188.188,-28.741,-43.006,179.814,5.698,149.064
C02560=1188.182,-28.491,-43.019,179.817,5.698,149.063
C02561=1188.177,-28.242,-43.032,179.819,5.698,149.062
C02562=1188.172,-27.992,-43.044,179.821,5.699,149.062
C02563=1188.167,-27.743,-43.056,179.824,5.699,149.061
C02564=1188.162,-27.492,-43.069,179.827,5.699,149.060
C02565=1188.157,-27.243,-43.082,179.829,5.700,149.060
C02566=1188.152,-26.994,-43.094,179.831,5.700,149.059
C02567=1188.146,-26.744,-43.106,179.834,5.700,149.058
C02568=1188.142,-26.494,-43.119,179.836,5.701,149.058
C02569=1188.136,-26.244,-43.132,179.839,5.701,149.057
C02570=1188.131,-25.995,-43.145,179.841,5.702,149.057
C02571=1188.126,-25.746,-43.158,179.844,5.703,149.056
C02572=1188.121,-25.496,-43.171,179.846,5.702,149.055
C02573=1188.116,-25.246,-43.183,179.848,5.703,149.055
C02574=1188.111,-24.996,-43.195,179.851,5.704,149.054
C02575=1188.105,-24.747,-43.208,179.853,5.704,149.053
C02576=1188.100,-24.497,-43.221,179.856,5.704,149.053
C02577=1188.095,-24.247,-43.234,179.858,5.704,149.052
C02578=1188.090,-23.998,-43.246,179.860,5.705,149.052
C02579=1188.084,-23.728,-43.261,179.863,5.705,149.051
C02580=1188.079,-23.459,-43.274,179.865,5.706,149.050
C02581=1188.074,-23.189,-43.288,179.868,5.706,149.049
C02582=1188.068,-22.919,-43.302,179.871,5.707,149.049
C02583=1188.063,-22.670,-43.315,179.873,5.707,149.048
C02584=1188.058,-22.421,-43.327,179.876,5.708,149.047
C02585=1188.053,-22.170,-43.341,179.879,5.708,149.047
C02586=1188.047,-21.921,-43.353,179.881,5.709,149.046
C02587=1188.042,-21.671,-43.365,179.883,5.709,149.045
C02588=1188.037,-21.422,-43.378,179.886,5.709,149.045
C02589=1188.032,-21.171,-43.391,179.888,5.710,149.044
C02590=1188.026,-20.922,-43.404,179.891,5.710,149.044
C02591=1188.021,-20.673,-43.417,179.893,5.711,149.043
C02592=1188.017,-20.423,-43.430,179.896,5.711,149.042
C02593=1188.011,-20.173,-43.443,179.898,5.711,149.042
C02594=1188.006,-19.924,-43.456,179.900,5.712,149.041
C02595=1188.002,-19.674,-43.469,179.903,5.712,149.040
C02596=1187.996,-19.425,-43.482,179.905,5.713,149.040
C02597=1187.991,-19.175,-43.495,179.908,5.713,149.039
C02598=1187.986,-18.925,-43.508,179.910,5.714,149.039
C02599=1187.980,-18.676,-43.521,179.913,5.715,149.038
C02600=1187.975,-18.426,-43.534,179.915,5.714,149.037
C02601=1187.971,-18.176,-43.547,179.918,5.715,149.036
C02602=1187.965,-17.927,-43.560,179.920,5.716,149.036
C02603=1187.960,-17.678,-43.572,179.922,5.716,149.035
C02604=1187.955,-17.427,-43.585,179.925,5.716,149.035
C02605=1187.949,-17.178,-43.599,179.928,5.717,149.034
C02606=1187.944,-16.929,-43.611,179.930,5.718,149.033
C02607=1187.940,-16.679,-43.625,179.932,5.717,149.033
C02608=1187.934,-16.430,-43.638,179.935,5.718,149.032
C02609=1187.929,-16.180,-43.651,179.937,5.718,149.031
C02610=1187.924,-15.930,-43.664,179.940,5.719,149.031
C02611=1187.919,-15.681,-43.677,179.942,5.720,149.030
C02612=1187.914,-15.431,-43.690,179.945,5.720,149.029
C02613=1187.909,-15.182,-43.703,179.947,5.721,149.029
C02614=1187.904,-14.932,-43.717,179.950,5.721,149.028
C02615=1187.899,-14.682,-43.729,179.952,5.721,149.028
C02616=1187.893,-14.433,-43.742,179.954,5.722,149.027
C02617=1187.888,-14.183,-43.755,179.957,5.722,149.026
C02618=1187.883,-13.934,-43.769,179.959,5.723,149.026
C02619=1187.878,-13.684,-43.782,179.962,5.723,149.025
C02620=1187.873,-13.434,-43.795,179.965,5.724,149.024
C02621=1187.867,-13.185,-43.808,179.967,5.724,149.024
C02622=1187.863,-12.935,-43.822,179.969,5.725,149.023
C02623=1187.857,-12.686,-43.835,179.971,5.725,149.023
C02624=1187.853,-12.436,-43.848,179.974,5.725,149.022
C02625=1187.847,-12.186,-43.861,179.977,5.726,149.021
C02626=1187.843,-11.936,-43.875,179.979,5.727,149.021
C02627=1187.837,-11.687,-43.888,179.982,5.727,149.020
C02628=1187.832,-11.437,-43.901,179.984,5.727,149.019
C02629=1187.827,-11.188,-43.914,179.987,5.728,149.019
C02630=1187.822,-10.939,-43.927,179.989,5.729,149.018
C02631=1187.817,-10.689,-43.940,179.992,5.729,149.017
C02632=1187.812,-10.440,-43.954,179.994,5.729,149.017
C02633=1187.807,-10.189,-43.967,179.996,5.729,149.016
C02634=1187.801,-9.940,-43.981,179.999,5.730,149.016
C02635=1187.797,-9.690,-43.994,-179.999,5.731,149.015
C02636=1187.791,-9.441,-44.007,-179.996,5.731,149.014
C02637=1187.787,-9.191,-44.020,-179.993,5.732,149.014
C02638=1187.781,-8.942,-44.034,-179.991,5.732,149.013
C02639=1187.776,-8.691,-44.048,-179.989,5.733,149.012
C02640=1187.771,-8.442,-44.060,-179.986,5.733,149.012
C02641=1187.766,-8.192,-44.075,-179.983,5.734,149.011
C02642=1187.761,-7.943,-44.087,-179.982,5.734,149.011
C02643=1187.756,-7.693,-44.102,-179.979,5.734,149.010
C02644=1187.750,-7.444,-44.114,-179.976,5.735,149.009
C02645=1187.745,-7.194,-44.128,-179.974,5.735,149.008
C02646=1187.740,-6.945,-44.141,-179.972,5.736,149.008
C02647=1187.735,-6.695,-44.155,-179.969,5.737,149.007
C02648=1187.730,-6.446,-44.169,-179.966,5.737,149.007
C02649=1187.725,-6.196,-44.182,-179.964,5.738,149.006
C02650=1187.719,-5.947,-44.195,-179.961,5.738,149.005
C02651=1187.715,-5.697,-44.208,-179.959,5.739,149.005
C02652=1187.710,-5.447,-44.223,-179.956,5.739,149.004
C02653=1187.704,-5.197,-44.236,-179.954,5.739,149.003
C02654=1187.700,-4.948,-44.250,-179.952,5.740,149.003
C02655=1187.694,-4.698,-44.263,-179.949,5.740,149.002
C02656=1187.690,-4.449,-44.276,-179.947,5.741,149.002
C02657=1187.684,-4.199,-44.290,-179.944,5.741,149.001
C02658=1187.679,-3.950,-44.304,-179.942,5.742,149.000
C02659=1187.674,-3.701,-44.317,-179.939,5.743,149.000
C02660=1187.669,-3.451,-44.331,-179.936,5.743,148.999
C02661=1187.664,-3.201,-44.345,-179.934,5.744,148.999
C02662=1187.659,-2.952,-44.358,-179.932,5.744,148.998
C02663=1187.654,-2.702,-44.372,-179.929,5.745,148.997
C02664=1187.648,-2.452,-44.385,-179.926,5.745,148.996
C02665=1187.644,-2.203,-44.399,-179.924,5.746,148.996
C02666=1187.639,-1.953,-44.413,-179.922,5.746,148.995
C02667=1187.633,-1.703,-44.426,-179.919,5.746,148.995
C02668=1187.629,-1.454,-44.440,-179.917,5.747,148.994
C02669=1187.623,-1.204,-44.453,-179.915,5.748,148.993
C02670=1187.618,-0.955,-44.467,-179.912,5.748,148.993
C02671=1187.613,-0.705,-44.482,-179.909,5.749,148.992
C02672=1187.608,-0.456,-44.494,-179.907,5.749,148.991
C02673=1187.603,-0.206,-44.509,-179.904,5.750,148.991
C02674=1187.597,0.043,-44.523,-179.902,5.750,148.990
C02675=1187.592,0.293,-44.536,-179.899,5.751,148.990
C02676=1187.588,0.543,-44.550,-179.896,5.751,148.989
C02677=1187.582,0.792,-44.564,-179.894,5.752,148.988
C02678=1187.577,1.042,-44.577,-179.892,5.753,148.988
C02679=1187.572,1.292,-44.592,-179.889,5.753,148.987
C02680=1187.567,1.541,-44.605,-179.886,5.754,148.986
C02681=1187.562,1.790,-44.619,-179.884,5.755,148.986
C02682=1187.556,2.040,-44.632,-179.882,5.755,148.985
C02683=1187.551,2.309,-44.647,-179.879,5.756,148.985
C02684=1187.546,2.578,-44.663,-179.876,5.756,148.984
C02685=1187.541,2.847,-44.678,-179.874,5.757,148.983
C02686=1187.535,3.117,-44.693,-179.871,5.757,148.982
C02687=1187.530,3.366,-44.706,-179.868,5.757,148.982
C02688=1187.525,3.616,-44.720,-179.866,5.758,148.981
C02689=1187.520,3.866,-44.734,-179.863,5.759,148.981
C02690=1187.514,4.115,-44.748,-179.861,5.759,148.980
C02691=1187.510,4.364,-44.762,-179.858,5.760,148.979
C02692=1187.505,4.614,-44.777,-179.856,5.761,148.979
C02693=1187.499,4.863,-44.789,-179.853,5.761,148.978
C02694=1187.494,5.113,-44.803,-179.851,5.762,148.977
C02695=1187.490,5.363,-44.818,-179.848,5.762,148.977
C02696=1187.485,5.613,-44.832,-179.846,5.763,148.976
C02697=1187.479,5.862,-44.846,-179.843,5.763,148.976
C02698=1187.474,6.111,-44.860,-179.841,5.764,148.975
C02699=1187.469,6.361,-44.875,-179.838,5.765,148.974
C02700=1187.463,6.611,-44.888,-179.836,5.765,148.974
C02701=1187.459,6.860,-44.901,-179.833,5.766,148.973
C02702=1187.454,7.110,-44.916,-179.830,5.766,148.972
C02703=1187.449,7.359,-44.930,-179.828,5.767,148.972
C02704=1187.444,7.608,-44.944,-179.826,5.767,148.971
C02705=1187.439,7.858,-44.958,-179.824,5.767,148.971
C02706=1187.434,8.108,-44.972,-179.821,5.768,148.970
C02707=1187.429,8.358,-44.987,-179.819,5.769,148.969
C02708=1187.423,8.607,-45.001,-179.816,5.769,148.969
C02709=1187.418,8.856,-45.015,-179.813,5.770,148.968
C02710=1187.413,9.106,-45.029,-179.811,5.770,148.968
C02711=1187.408,9.356,-45.043,-179.809,5.771,148.967
C02712=1187.403,9.605,-45.057,-179.806,5.771,148.966
C02713=1187.398,9.854,-45.072,-179.803,5.772,148.966
C02714=1187.393,10.104,-45.086,-179.801,5.773,148.965
C02715=1187.388,10.354,-45.100,-179.798,5.773,148.964
C02716=1187.383,10.604,-45.114,-179.796,5.774,148.964
C02717=1187.377,10.853,-45.128,-179.793,5.774,148.963
C02718=1187.372,11.102,-45.143,-179.791,5.775,148.963
C02719=1187.367,11.352,-45.157,-179.788,5.775,148.962
C02720=1187.362,11.602,-45.171,-179.786,5.776,148.961
C02721=1187.358,11.851,-45.185,-179.784,5.777,148.961
C02722=1187.352,12.100,-45.199,-179.781,5.777,148.960
C02723=1187.347,12.350,-45.214,-179.778,5.778,148.959
C02724=1187.342,12.600,-45.228,-179.776,5.778,148.959
C02725=1187.337,12.850,-45.242,-179.773,5.779,148.958
C02726=1187.332,13.099,-45.256,-179.771,5.780,148.958
C02727=1187.327,13.349,-45.271,-179.768,5.780,148.957
C02728=1187.322,13.597,-45.285,-179.766,5.781,148.956
C02729=1187.317,13.847,-45.300,-179.763,5.781,148.956
C02730=1187.312,14.097,-45.314,-179.761,5.782,148.955
C02731=1187.307,14.346,-45.328,-179.758,5.782,148.954
C02732=1187.302,14.596,-45.342,-179.756,5.783,148.954
C02733=1187.297,14.846,-45.357,-179.753,5.785,148.953
C02734=1187.292,15.095,-45.371,-179.750,5.785,148.953
C02735=1187.287,15.344,-45.386,-179.747,5.786,148.952
C02736=1187.282,15.594,-45.400,-179.745,5.786,148.951
C02737=1187.276,15.844,-45.415,-179.743,5.787,148.951
C02738=1187.271,16.093,-45.429,-179.740,5.787,148.950
C02739=1187.266,16.343,-45.443,-179.738,5.788,148.950
C02740=1187.262,16.592,-45.458,-179.735,5.789,148.949
C02741=1187.257,16.842,-45.473,-179.732,5.789,148.948
C02742=1187.251,17.091,-45.487,-179.730,5.790,148.948
C02743=1187.246,17.341,-45.501,-179.728,5.791,148.947
C02744=1187.242,17.590,-45.516,-179.725,5.791,148.946
C02745=1187.236,17.840,-45.531,-179.722,5.792,148.946
C02746=1187.231,18.089,-45.545,-179.720,5.792,148.945
C02747=1187.226,18.339,-45.559,-179.717,5.793,148.945
C02748=1187.221,18.588,-45.574,-179.715,5.793,148.944
C02749=1187.216,18.838,-45.589,-179.712,5.794,148.943
C02750=1187.211,19.088,-45.603,-179.710,5.795,148.943
C02751=1187.206,19.337,-45.618,-179.707,5.795,148.942
C02752=1187.201,19.587,-45.633,-179.705,5.796,148.941
C02753=1187.196,19.836,-45.647,-179.703,5.797,148.941
C02754=1187.191,20.085,-45.662,-179.700,5.797,148.940
C02755=1187.186,20.335,-45.676,-179.697,5.798,148.940
C02756=1187.180,20.585,-45.691,-179.695,5.798,148.939
C02757=1187.176,20.834,-45.706,-179.692,5.799,148.938
C02758=1187.171,21.083,-45.720,-179.690,5.800,148.938
C02759=1187.166,21.333,-45.734,-179.687,5.800,148.937
C02760=1187.160,21.583,-45.750,-179.685,5.801,148.937
C02761=1187.155,21.832,-45.764,-179.682,5.802,148.936
C02762=1187.150,22.082,-45.778,-179.679,5.803,148.935
C02763=1187.146,22.331,-45.793,-179.677,5.804,148.935
C02764=1187.140,22.581,-45.808,-179.674,5.804,148.934
C02765=1187.135,22.830,-45.823,-179.672,5.805,148.933
C02766=1187.131,23.080,-45.838,-179.669,5.805,148.933
C02767=1187.126,23.329,-45.853,-179.667,5.806,148.932
C02768=1187.120,23.579,-45.867,-179.664,5.806,148.932
C02769=1187.116,23.828,-45.882,-179.662,5.807,148.931
C02770=1187.111,24.078,-45.897,-179.659,5.808,148.931
C02771=1187.105,24.327,-45.912,-179.657,5.808,148.930
C02772=1187.100,24.577,-45.927,-179.654,5.809,148.929
C02773=1187.095,24.827,-45.941,-179.652,5.810,148.929
C02774=1187.090,25.076,-45.956,-179.649,5.810,148.928
C02775=1187.085,25.325,-45.971,-179.647,5.811,148.927
C02776=1187.080,25.575,-45.986,-179.643,5.812,148.927
C02777=1187.075,25.824,-46.001,-179.641,5.813,148.926
C02778=1187.070,26.074,-46.016,-179.639,5.813,148.926
C02779=1187.065,26.323,-46.031,-179.636,5.814,148.925
C02780=1187.060,26.573,-46.045,-179.634,5.815,148.924
C02781=1187.055,26.822,-46.060,-179.631,5.815,148.924
C02782=1187.050,27.072,-46.075,-179.629,5.816,148.923
C02783=1187.045,27.321,-46.090,-179.626,5.817,148.923
C02784=1187.040,27.570,-46.105,-179.624,5.817,148.922
C02785=1187.034,27.820,-46.120,-179.621,5.818,148.921
C02786=1187.030,28.069,-46.135,-179.618,5.818,148.921
C02787=1187.024,28.338,-46.151,-179.616,5.820,148.920
C02788=1187.019,28.607,-46.167,-179.613,5.820,148.919
C02789=1187.013,28.876,-46.183,-179.610,5.821,148.919
C02790=1187.008,29.145,-46.200,-179.608,5.821,148.918
C02791=1187.003,29.394,-46.214,-179.605,5.822,148.917
C02792=1186.998,29.644,-46.230,-179.602,5.823,148.917
C02793=1186.994,29.894,-46.245,-179.600,5.824,148.916
C02794=1186.988,30.144,-46.260,-179.597,5.824,148.916
C02795=1186.983,30.393,-46.275,-179.594,5.825,148.915
C02796=1186.978,30.642,-46.291,-179.592,5.826,148.914
C02797=1186.973,30.892,-46.305,-179.590,5.826,148.914
C02798=1186.968,31.141,-46.320,-179.587,5.827,148.913
C02799=1186.963,31.390,-46.335,-179.585,5.828,148.913
C02800=1186.958,31.639,-46.350,-179.582,5.828,148.912
C02801=1186.953,31.890,-46.366,-179.579,5.829,148.911
C02802=1186.948,32.139,-46.381,-179.577,5.830,148.911
C02803=1186.943,32.389,-46.396,-179.574,5.831,148.910
C02804=1186.938,32.638,-46.411,-179.571,5.831,148.910
C02805=1186.933,32.888,-46.426,-179.569,5.832,148.909
C02806=1186.928,33.137,-46.441,-179.567,5.833,148.908
C02807=1186.923,33.386,-46.457,-179.564,5.833,148.908
C02808=1186.918,33.635,-46.472,-179.562,5.834,148.907
C02809=1186.913,33.885,-46.488,-179.559,5.835,148.907
C02810=1186.908,34.135,-46.502,-179.556,5.836,148.906
C02811=1186.903,34.385,-46.517,-179.554,5.837,148.905
C02812=1186.898,34.634,-46.533,-179.551,5.837,148.905
C02813=1186.893,34.883,-46.548,-179.549,5.838,148.904
C02814=1186.887,35.132,-46.564,-179.546,5.838,148.903
C02815=1186.883,35.382,-46.579,-179.544,5.839,148.903
C02816=1186.878,35.632,-46.594,-179.541,5.840,148.902
C02817=1186.872,35.882,-46.609,-179.538,5.840,148.902
C02818=1186.868,36.131,-46.624,-179.536,5.842,148.901
C02819=1186.862,36.380,-46.640,-179.533,5.842,148.901
C02820=1186.858,36.630,-46.655,-179.530,5.843,148.900
C02821=1186.853,36.879,-46.671,-179.528,5.844,148.899
C02822=1186.847,37.129,-46.687,-179.526,5.844,148.899
C02823=1186.843,37.378,-46.702,-179.523,5.845,148.898
C02824=1186.837,37.627,-46.717,-179.521,5.846,148.898
C02825=1186.833,37.877,-46.733,-179.518,5.847,148.897
C02826=1186.828,38.126,-46.748,-179.515,5.847,148.896
C02827=1186.823,38.376,-46.764,-179.513,5.848,148.896
C02828=1186.818,38.625,-46.779,-179.510,5.849,148.895
C02829=1186.813,38.875,-46.795,-179.508,5.849,148.894
C02830=1186.808,39.124,-46.810,-179.505,5.850,148.894
C02831=1186.803,39.373,-46.825,-179.503,5.851,148.893
C02832=1186.798,39.623,-46.841,-179.500,5.852,148.893
C02833=1186.792,39.872,-46.856,-179.497,5.853,148.892
C02834=1186.788,40.122,-46.872,-179.495,5.853,148.892
C02835=1186.783,40.371,-46.887,-179.492,5.854,148.891
C02836=1186.778,40.621,-46.903,-179.490,5.855,148.890
C02837=1186.773,40.871,-46.919,-179.487,5.855,148.890
C02838=1186.768,41.120,-46.934,-179.484,5.857,148.889
C02839=1186.763,41.369,-46.949,-179.482,5.858,148.889
C02840=1186.757,41.619,-46.965,-179.479,5.858,148.888
C02841=1186.753,41.869,-46.981,-179.477,5.859,148.888
C02842=1186.748,42.118,-46.996,-179.474,5.859,148.887
C02843=1186.743,42.367,-47.012,-179.472,5.860,148.886
C02844=1186.737,42.617,-47.027,-179.469,5.862,148.886
C02845=1186.732,42.867,-47.043,-179.466,5.862,148.885
C02846=1186.728,43.115,-47.059,-179.464,5.863,148.884
C02847=1186.723,43.365,-47.074,-179.462,5.864,148.884
C02848=1186.718,43.615,-47.090,-179.459,5.864,148.883
C02849=1186.712,43.864,-47.106,-179.456,5.865,148.883
C02850=1186.708,44.113,-47.121,-179.454,5.866,148.882
C02851=1186.703,44.364,-47.137,-179.451,5.867,148.881
C02852=1186.698,44.612,-47.153,-179.448,5.867,148.881
C02853=1186.693,44.862,-47.169,-179.446,5.868,148.880
C02854=1186.688,45.112,-47.185,-179.444,5.869,148.880
C02855=1186.682,45.361,-47.200,-179.441,5.869,148.879
C02856=1186.678,45.610,-47.215,-179.438,5.871,148.879
C02857=1186.673,45.860,-47.232,-179.436,5.871,148.878
C02858=1186.668,46.109,-47.248,-179.433,5.872,148.877
C02859=1186.662,46.359,-47.263,-179.431,5.873,148.877
C02860=1186.658,46.609,-47.279,-179.428,5.873,148.876
C02861=1186.653,46.858,-47.295,-179.425,5.875,148.876
C02862=1186.648,47.107,-47.310,-179.423,5.876,148.875
C02863=1186.643,47.357,-47.326,-179.420,5.876,148.874
C02864=1186.638,47.605,-47.343,-179.418,5.877,148.874
C02865=1186.633,47.856,-47.359,-179.415,5.877,148.873
C02866=1186.628,48.105,-47.374,-179.412,5.879,148.873
C02867=1186.623,48.354,-47.390,-179.410,5.880,148.872
C02868=1186.618,48.604,-47.406,-179.407,5.880,148.871
C02869=1186.613,48.853,-47.422,-179.405,5.881,148.871
C02870=1186.608,49.103,-47.438,-179.403,5.882,148.870
C02871=1186.604,49.352,-47.454,-179.399,5.883,148.870
C02872=1186.598,49.601,-47.469,-179.397,5.884,148.869
C02873=1186.594,49.851,-47.486,-179.395,5.884,148.869
C02874=1186.588,50.100,-47.502,-179.392,5.885,148.868
C02875=1186.583,50.350,-47.518,-179.390,5.886,148.867
C02876=1186.578,50.599,-47.534,-179.387,5.887,148.867
C02877=1186.574,50.849,-47.550,-179.384,5.888,148.866
C02878=1186.569,51.098,-47.566,-179.382,5.888,148.866
C02879=1186.563,51.347,-47.582,-179.379,5.889,148.865
C02880=1186.558,51.597,-47.598,-179.376,5.890,148.864
C02881=1186.553,51.846,-47.614,-179.374,5.891,148.864
C02882=1186.549,52.096,-47.630,-179.371,5.892,148.863
C02883=1186.543,52.345,-47.646,-179.369,5.893,148.863
C02884=1186.539,52.595,-47.662,-179.366,5.893,148.862
C02885=1186.534,52.844,-47.678,-179.363,5.894,148.861
C02886=1186.529,53.094,-47.694,-179.361,5.895,148.861
C02887=1186.524,53.343,-47.711,-179.358,5.896,148.860
C02888=1186.519,53.593,-47.727,-179.356,5.896,148.860
C02889=1186.514,53.842,-47.743,-179.353,5.898,148.859
C02890=1186.509,54.092,-47.759,-179.350,5.899,148.859
C02891=1186.504,54.360,-47.777,-179.348,5.899,148.858
C02892=1186.498,54.628,-47.794,-179.345,5.901,148.858
C02893=1186.493,54.897,-47.811,-179.342,5.901,148.857
C02894=1186.488,55.165,-47.829,-179.340,5.902,148.856
C02895=1186.482,55.415,-47.845,-179.336,5.903,148.856
C02896=1186.477,55.664,-47.862,-179.334,5.904,148.855
C02897=1186.472,55.914,-47.877,-179.332,5.905,148.854
C02898=1186.468,56.163,-47.894,-179.330,5.906,148.854
C02899=1186.462,56.412,-47.910,-179.326,5.907,148.853
C02900=1186.458,56.662,-47.926,-179.324,5.907,148.853
C02901=1186.453,56.911,-47.942,-179.321,5.908,148.852
C02902=1186.448,57.161,-47.958,-179.319,5.909,148.852
C02903=1186.443,57.410,-47.975,-179.316,5.911,148.851
C02904=1186.438,57.660,-47.992,-179.313,5.911,148.850
C02905=1186.433,57.910,-48.008,-179.311,5.912,148.850
C02906=1186.428,58.159,-48.024,-179.309,5.912,148.849
C02907=1186.423,58.408,-48.041,-179.305,5.914,148.849
C02908=1186.418,58.657,-48.056,-179.303,5.914,148.848
C02909=1186.413,58.907,-48.073,-179.301,5.915,148.848
C02910=1186.408,59.156,-48.089,-179.297,5.917,148.847
C02911=1186.403,59.406,-48.107,-179.295,5.917,148.846
C02912=1186.398,59.655,-48.122,-179.293,5.918,148.846
C02913=1186.393,59.904,-48.139,-179.290,5.918,148.845
C02914=1186.389,60.154,-48.156,-179.287,5.920,148.845
C02915=1186.384,60.403,-48.172,-179.285,5.921,148.844
C02916=1186.378,60.653,-48.188,-179.283,5.922,148.844
C02917=1186.373,60.902,-48.205,-179.280,5.922,148.843
C02918=1186.368,61.151,-48.221,-179.277,5.924,148.843
C02919=1186.364,61.401,-48.238,-179.275,5.924,148.842
C02920=1186.359,61.650,-48.254,-179.272,5.925,148.841
C02921=1186.353,61.900,-48.271,-179.269,5.927,148.841
C02922=1186.348,62.149,-48.287,-179.267,5.927,148.840
C02923=1186.344,62.398,-48.304,-179.264,5.928,148.840
C02924=1186.339,62.648,-48.321,-179.262,5.929,148.839
C02925=1186.334,62.897,-48.338,-179.259,5.930,148.838
C02926=1186.329,63.147,-48.353,-179.256,5.931,148.838
C02927=1186.324,63.396,-48.370,-179.254,5.931,148.837
C02928=1186.318,63.646,-48.387,-179.251,5.933,148.837
C02929=1186.314,63.895,-48.404,-179.248,5.934,148.836
C02930=1186.309,64.144,-48.420,-179.246,5.934,148.835
C02931=1186.304,64.393,-48.437,-179.244,5.935,148.835
C02932=1186.299,64.643,-48.454,-179.240,5.936,148.834
C02933=1186.294,64.892,-48.470,-179.238,5.937,148.834
C02934=1186.290,65.141,-48.487,-179.236,5.938,148.833
C02935=1186.284,65.391,-48.504,-179.233,5.939,148.833
C02936=1186.279,65.640,-48.520,-179.230,5.940,148.832
C02937=1186.275,65.890,-48.536,-179.228,5.940,148.832
C02938=1186.269,66.140,-48.554,-179.225,5.942,148.831
C02939=1186.265,66.389,-48.570,-179.222,5.943,148.830
C02940=1186.260,66.638,-48.587,-179.220,5.944,148.830
C02941=1186.255,66.888,-48.604,-179.218,5.944,148.829
C02942=1186.250,67.137,-48.621,-179.215,5.946,148.829
C02943=1186.245,67.386,-48.637,-179.212,5.946,148.828
C02944=1186.240,67.636,-48.654,-179.210,5.947,148.828
C02945=1186.235,67.885,-48.671,-179.207,5.949,148.827
C02946=1186.230,68.135,-48.689,-179.204,5.949,148.826
C02947=1186.225,68.383,-48.705,-179.202,5.950,148.826
C02948=1186.221,68.633,-48.722,-179.199,5.951,148.825
C02949=1186.216,68.883,-48.739,-179.197,5.952,148.825
C02950=1186.211,69.131,-48.755,-179.194,5.953,148.824
C02951=1186.205,69.381,-48.773,-179.191,5.954,148.824
C02952=1186.201,69.631,-48.789,-179.189,5.955,148.823
C02953=1186.196,69.881,-48.807,-179.186,5.956,148.823
C02954=1186.191,70.129,-48.823,-179.183,5.957,148.822
C02955=1186.186,70.379,-48.840,-179.181,5.958,148.821
C02956=1186.181,70.629,-48.857,-179.179,5.959,148.821
C02957=1186.177,70.877,-48.874,-179.175,5.960,148.820
C02958=1186.171,71.127,-48.891,-179.173,5.961,148.820
C02959=1186.166,71.376,-48.908,-179.171,5.962,148.819
C02960=1186.161,71.626,-48.925,-179.167,5.963,148.819
C02961=1186.157,71.875,-48.942,-179.165,5.964,148.818
C02962=1186.151,72.125,-48.959,-179.163,5.964,148.818
C02963=1186.147,72.373,-48.976,-179.160,5.966,148.817
C02964=1186.141,72.623,-48.993,-179.157,5.967,148.816
C02965=1186.137,72.873,-49.010,-179.155,5.967,148.816
C02966=1186.132,73.122,-49.027,-179.152,5.969,148.815
C02967=1186.127,73.372,-49.044,-179.150,5.970,148.815
C02968=1186.122,73.620,-49.061,-179.147,5.970,148.814
C02969=1186.117,73.870,-49.078,-179.144,5.972,148.814
C02970=1186.112,74.120,-49.095,-179.142,5.973,148.813
C02971=1186.107,74.369,-49.113,-179.139,5.973,148.813
C02972=1186.103,74.618,-49.130,-179.136,5.975,148.812
C02973=1186.097,74.867,-49.147,-179.134,5.975,148.811
C02974=1186.092,75.117,-49.164,-179.131,5.977,148.811
C02975=1186.087,75.366,-49.182,-179.128,5.978,148.810
C02976=1186.083,75.616,-49.198,-179.126,5.978,148.810
C02977=1186.078,75.865,-49.216,-179.123,5.980,148.809
C02978=1186.073,76.114,-49.234,-179.121,5.981,148.809
C02979=1186.068,76.364,-49.250,-179.118,5.981,148.808
C02980=1186.063,76.613,-49.267,-179.116,5.983,148.808
C02981=1186.058,76.862,-49.285,-179.113,5.984,148.807
C02982=1186.053,77.112,-49.302,-179.111,5.984,148.807
C02983=1186.048,77.361,-49.320,-179.108,5.986,148.806
C02984=1186.044,77.610,-49.336,-179.105,5.986,148.805
C02985=1186.039,77.860,-49.354,-179.102,5.988,148.805
C02986=1186.034,78.109,-49.372,-179.100,5.989,148.804
C02987=1186.029,78.359,-49.388,-179.098,5.989,148.804
C02988=1186.024,78.607,-49.406,-179.094,5.991,148.803
C02989=1186.018,78.857,-49.423,-179.092,5.992,148.803
C02990=1186.014,79.107,-49.440,-179.089,5.993,148.802
C02991=1186.009,79.356,-49.458,-179.087,5.994,148.802
C02992=1186.004,79.606,-49.475,-179.084,5.995,148.801
C02993=1185.999,79.855,-49.493,-179.081,5.996,148.801
C02994=1185.994,80.104,-49.510,-179.079,5.997,148.800
C02995=1185.989,80.372,-49.529,-179.076,5.998,148.800
C02996=1185.983,80.641,-49.547,-179.074,5.999,148.799
C02997=1185.978,80.909,-49.567,-179.070,6.000,148.798
C02998=1185.974,81.177,-49.585,-179.068,6.001,148.798
C02999=1185.969,81.427,-49.603,-179.065,6.003,148.797
C03000=1185.963,81.676,-49.620,-179.062,6.003,148.797
C03001=1185.959,81.926,-49.638,-179.060,6.005,148.796
C03002=1185.954,82.175,-49.655,-179.057,6.005,148.795
C03003=1185.949,82.424,-49.673,-179.055,6.006,148.795
C03004=1185.944,82.674,-49.690,-179.052,6.008,148.794
C03005=1185.939,82.923,-49.708,-179.049,6.009,148.794
C03006=1185.934,83.172,-49.726,-179.046,6.010,148.793
C03007=1185.929,83.421,-49.742,-179.044,6.011,148.793
C03008=1185.924,83.670,-49.760,-179.042,6.011,148.792
C03009=1185.919,83.920,-49.778,-179.039,6.013,148.792
C03010=1185.914,84.169,-49.796,-179.036,6.014,148.791
C03011=1185.909,84.419,-49.814,-179.033,6.015,148.791
C03012=1185.905,84.668,-49.830,-179.031,6.016,148.790
C03013=1185.900,84.917,-49.848,-179.028,6.018,148.790
C03014=1185.895,85.166,-49.866,-179.025,6.018,148.789
C03015=1185.890,85.416,-49.883,-179.023,6.019,148.789
C03016=1185.885,85.665,-49.901,-179.020,6.021,148.788
C03017=1185.880,85.914,-49.919,-179.018,6.021,148.788
C03018=1185.875,86.164,-49.938,-179.015,6.023,148.787
C03019=1185.871,86.414,-49.954,-179.013,6.024,148.786
C03020=1185.866,86.663,-49.972,-179.009,6.025,148.786
C03021=1185.861,86.912,-49.990,-179.007,6.026,148.785
C03022=1185.856,87.161,-50.008,-179.005,6.027,148.785
C03023=1185.851,87.411,-50.026,-179.002,6.028,148.784
C03024=1185.846,87.660,-50.044,-178.999,6.029,148.784
C03025=1185.841,87.910,-50.062,-178.997,6.031,148.783
C03026=1185.836,88.159,-50.080,-178.995,6.031,148.783
C03027=1185.831,88.409,-50.097,-178.991,6.033,148.782
C03028=1185.826,88.658,-50.115,-178.989,6.034,148.782
C03029=1185.821,88.907,-50.133,-178.987,6.034,148.781
C03030=1185.817,89.156,-50.150,-178.984,6.036,148.781
C03031=1185.812,89.405,-50.168,-178.981,6.037,148.780
C03032=1185.807,89.654,-50.186,-178.979,6.038,148.780
C03033=1185.802,89.904,-50.203,-178.976,6.039,148.779
C03034=1185.797,90.153,-50.221,-178.973,6.041,148.779
C03035=1185.793,90.403,-50.240,-178.971,6.041,148.778
C03036=1185.788,90.652,-50.258,-178.968,6.043,148.777
C03037=1185.783,90.901,-50.276,-178.965,6.043,148.777
C03038=1185.778,91.150,-50.294,-178.962,6.045,148.776
C03039=1185.773,91.400,-50.312,-178.960,6.046,148.776
C03040=1185.768,91.649,-50.330,-178.958,6.047,148.775
C03041=1185.763,91.898,-50.348,-178.955,6.048,148.775
C03042=1185.758,92.147,-50.366,-178.952,6.049,148.774
C03043=1185.754,92.396,-50.384,-178.950,6.051,148.774
C03044=1185.749,92.646,-50.402,-178.947,6.051,148.773
C03045=1185.744,92.895,-50.420,-178.944,6.053,148.773
C03046=1185.739,93.145,-50.438,-178.942,6.053,148.772
C03047=1185.734,93.394,-50.456,-178.939,6.055,148.772
C03048=1185.729,93.643,-50.474,-178.936,6.056,148.771
C03049=1185.724,93.892,-50.492,-178.934,6.057,148.771
C03050=1185.720,94.142,-50.511,-178.931,6.058,148.770
C03051=1185.715,94.391,-50.529,-178.928,6.060,148.770
C03052=1185.710,94.641,-50.547,-178.926,6.060,148.769
C03053=1185.705,94.890,-50.565,-178.923,6.062,148.769
C03054=1185.700,95.139,-50.583,-178.921,6.063,148.768
C03055=1185.695,95.388,-50.601,-178.918,6.064,148.767
C03056=1185.691,95.638,-50.619,-178.916,6.065,148.767
C03057=1185.685,95.888,-50.638,-178.912,6.066,148.766
C03058=1185.680,96.137,-50.656,-178.910,6.067,148.766
C03059=1185.675,96.386,-50.674,-178.907,6.069,148.765
C03060=1185.670,96.635,-50.692,-178.905,6.070,148.765
C03061=1185.666,96.884,-50.711,-178.902,6.071,148.764
C03062=1185.661,97.133,-50.729,-178.900,6.072,148.764
C03063=1185.657,97.383,-50.747,-178.897,6.074,148.763
C03064=1185.651,97.632,-50.765,-178.894,6.074,148.763
C03065=1185.646,97.881,-50.783,-178.891,6.076,148.762
C03066=1185.642,98.131,-50.801,-178.889,6.077,148.762
C03067=1185.637,98.380,-50.820,-178.886,6.078,148.761
C03068=1185.632,98.629,-50.838,-178.884,6.079,148.761
C03069=1185.626,98.878,-50.857,-178.881,6.081,148.760
C03070=1185.622,99.128,-50.875,-178.879,6.081,148.760
C03071=1185.617,99.377,-50.893,-178.876,6.083,148.759
C03072=1185.613,99.626,-50.912,-178.873,6.084,148.759
C03073=1185.607,99.875,-50.930,-178.870,6.085,148.758
C03074=1185.603,100.125,-50.949,-178.868,6.086,148.758
C03075=1185.598,100.375,-50.967,-178.865,6.087,148.757
C03076=1185.593,100.623,-50.985,-178.863,6.088,148.757
C03077=1185.588,100.873,-51.004,-178.860,6.090,148.756
C03078=1185.583,101.122,-51.022,-178.857,6.091,148.756
C03079=1185.579,101.371,-51.041,-178.855,6.092,148.755
C03080=1185.574,101.620,-51.059,-178.852,6.093,148.755
C03081=1185.569,101.870,-51.078,-178.849,6.095,148.754
C03082=1185.564,102.119,-51.097,-178.847,6.096,148.754
C03083=1185.559,102.368,-51.115,-178.844,6.097,148.753
C03084=1185.554,102.618,-51.133,-178.842,6.098,148.753
C03085=1185.549,102.867,-51.152,-178.839,6.099,148.752
C03086=1185.545,103.116,-51.170,-178.837,6.100,148.752
C03087=1185.540,103.365,-51.188,-178.833,6.102,148.751
C03088=1185.535,103.615,-51.208,-178.831,6.103,148.751
C03089=1185.530,103.864,-51.226,-178.829,6.104,148.750
C03090=1185.525,104.113,-51.245,-178.825,6.106,148.750
C03091=1185.520,104.363,-51.263,-178.823,6.107,148.749
C03092=1185.516,104.611,-51.282,-178.820,6.108,148.749
C03093=1185.511,104.861,-51.301,-178.818,6.109,148.748
C03094=1185.506,105.111,-51.319,-178.815,6.111,148.748
C03095=1185.501,105.359,-51.338,-178.813,6.111,148.747
C03096=1185.496,105.609,-51.357,-178.810,6.113,148.747
C03097=1185.491,105.858,-51.375,-178.807,6.113,148.746
C03098=1185.486,106.107,-51.394,-178.805,6.115,148.746
C03099=1185.482,106.376,-51.414,-178.802,6.117,148.745
C03100=1185.476,106.644,-51.434,-178.799,6.118,148.745
C03101=1185.471,106.912,-51.455,-178.796,6.119,148.744
C03102=1185.466,107.181,-51.475,-178.793,6.121,148.744
C03103=1185.461,107.430,-51.494,-178.790,6.122,148.743
C03104=1185.456,107.679,-51.512,-178.788,6.123,148.742
C03105=1185.452,107.929,-51.531,-178.785,6.125,148.742
C03106=1185.446,108.178,-51.550,-178.783,6.125,148.741
C03107=1185.442,108.427,-51.569,-178.780,6.127,148.741
C03108=1185.437,108.676,-51.588,-178.778,6.128,148.741
C03109=1185.432,108.925,-51.606,-178.775,6.129,148.740
C03110=1185.427,109.175,-51.626,-178.772,6.131,148.740
C03111=1185.422,109.424,-51.644,-178.769,6.132,148.739
C03112=1185.417,109.674,-51.663,-178.767,6.133,148.739
C03113=1185.413,109.922,-51.682,-178.764,6.134,148.738
C03114=1185.408,110.172,-51.701,-178.761,6.136,148.737
C03115=1185.403,110.421,-51.720,-178.759,6.136,148.737
C03116=1185.398,110.670,-51.739,-178.756,6.138,148.737
C03117=1185.393,110.920,-51.757,-178.753,6.140,148.736
C03118=1185.388,111.169,-51.777,-178.751,6.141,148.736
C03119=1185.384,111.418,-51.796,-178.748,6.142,148.735
C03120=1185.378,111.667,-51.814,-178.746,6.143,148.735
C03121=1185.374,111.917,-51.833,-178.743,6.145,148.734
C03122=1185.369,112.165,-51.853,-178.740,6.146,148.734
C03123=1185.364,112.415,-51.872,-178.738,6.147,148.733
C03124=1185.359,112.664,-51.890,-178.735,6.149,148.733
C03125=1185.355,112.914,-51.910,-178.732,6.149,148.732
C03126=1185.350,113.162,-51.929,-178.730,6.151,148.732
C03127=1185.345,113.412,-51.948,-178.727,6.153,148.731
C03128=1185.340,113.661,-51.968,-178.724,6.153,148.731
C03129=1185.336,113.911,-51.986,-178.722,6.155,148.730
C03130=1185.330,114.159,-52.005,-178.720,6.156,148.730
C03131=1185.326,114.409,-52.025,-178.716,6.157,148.729
C03132=1185.321,114.658,-52.044,-178.714,6.159,148.729
C03133=1185.316,114.907,-52.063,-178.712,6.160,148.728
C03134=1185.312,115.156,-52.082,-178.708,6.161,148.728
C03135=1185.307,115.406,-52.101,-178.706,6.162,148.727
C03136=1185.301,115.655,-52.120,-178.703,6.164,148.727
C03137=1185.296,115.904,-52.140,-178.700,6.165,148.726
C03138=1185.292,116.153,-52.159,-178.698,6.166,148.726
C03139=1185.287,116.402,-52.178,-178.695,6.168,148.725
C03140=1185.282,116.652,-52.198,-178.692,6.169,148.725
C03141=1185.278,116.901,-52.217,-178.690,6.170,148.724
C03142=1185.273,117.150,-52.236,-178.687,6.172,148.724
C03143=1185.268,117.399,-52.255,-178.685,6.173,148.723
C03144=1185.264,117.648,-52.275,-178.682,6.174,148.723
C03145=1185.258,117.897,-52.294,-178.679,6.176,148.722
C03146=1185.254,118.147,-52.314,-178.677,6.177,148.722
C03147=1185.249,118.396,-52.333,-178.674,6.178,148.722
C03148=1185.244,118.645,-52.352,-178.672,6.180,148.721
C03149=1185.239,118.894,-52.372,-178.669,6.181,148.721
C03150=1185.234,119.143,-52.391,-178.666,6.183,148.720
C03151=1185.229,119.393,-52.410,-178.663,6.184,148.720
C03152=1185.225,119.642,-52.430,-178.661,6.185,148.719
C03153=1185.220,119.891,-52.449,-178.658,6.187,148.719
C03154=1185.215,120.141,-52.468,-178.656,6.188,148.718
C03155=1185.210,120.389,-52.488,-178.653,6.189,148.718
C03156=1185.205,120.639,-52.507,-178.650,6.191,148.717
C03157=1185.201,120.888,-52.526,-178.648,6.192,148.717
C03158=1185.196,121.137,-52.546,-178.645,6.193,148.716
C03159=1185.191,121.387,-52.565,-178.642,6.195,148.716
C03160=1185.186,121.636,-52.585,-178.640,6.196,148.715
C03161=1185.181,121.884,-52.605,-178.637,6.197,148.715
C03162=1185.177,122.134,-52.625,-178.634,6.199,148.714
C03163=1185.173,122.383,-52.644,-178.632,6.200,148.714
C03164=1185.167,122.632,-52.663,-178.629,6.202,148.714
C03165=1185.162,122.882,-52.683,-178.626,6.203,148.713
C03166=1185.158,123.131,-52.702,-178.624,6.204,148.713
C03167=1185.153,123.380,-52.722,-178.621,6.206,148.712
C03168=1185.148,123.629,-52.742,-178.618,6.207,148.712
C03169=1185.143,123.879,-52.762,-178.616,6.208,148.711
C03170=1185.138,124.128,-52.781,-178.613,6.210,148.711
C03171=1185.133,124.377,-52.801,-178.610,6.211,148.710
C03172=1185.129,124.626,-52.820,-178.608,6.212,148.710
C03173=1185.124,124.875,-52.840,-178.605,6.214,148.709
C03174=1185.119,125.124,-52.859,-178.603,6.215,148.709
C03175=1185.115,125.373,-52.880,-178.600,6.216,148.708
C03176=1185.110,125.623,-52.899,-178.597,6.218,148.708
C03177=1185.105,125.872,-52.919,-178.595,6.220,148.708
C03178=1185.100,126.121,-52.938,-178.592,6.220,148.707
C03179=1185.096,126.370,-52.959,-178.589,6.222,148.707
C03180=1185.090,126.619,-52.978,-178.587,6.224,148.706
C03181=1185.086,126.869,-52.998,-178.584,6.225,148.706
C03182=1185.081,127.117,-53.018,-178.581,6.226,148.705
C03183=1185.076,127.367,-53.038,-178.579,6.228,148.705
C03184=1185.071,127.616,-53.057,-178.576,6.229,148.704
C03185=1185.067,127.865,-53.077,-178.574,6.230,148.704
C03186=1185.062,128.114,-53.097,-178.571,6.232,148.703
C03187=1185.057,128.363,-53.117,-178.568,6.234,148.703
C03188=1185.053,128.613,-53.137,-178.566,6.234,148.702
C03189=1185.047,128.862,-53.156,-178.563,6.236,148.702
C03190=1185.043,129.111,-53.177,-178.560,6.238,148.701
C03191=1185.038,129.360,-53.196,-178.557,6.239,148.701
C03192=1185.034,129.609,-53.217,-178.555,6.240,148.701
C03193=1185.028,129.858,-53.236,-178.552,6.242,148.700
C03194=1185.024,130.107,-53.256,-178.549,6.243,148.700
C03195=1185.019,130.357,-53.276,-178.547,6.244,148.699
C03196=1185.015,130.606,-53.296,-178.544,6.246,148.699
C03197=1185.009,130.855,-53.317,-178.541,6.248,148.698
C03198=1185.004,131.104,-53.337,-178.538,6.249,148.698
C03199=1184.999,131.353,-53.356,-178.536,6.250,148.697
C03200=1184.995,131.602,-53.377,-178.534,6.252,148.697
C03201=1184.990,131.852,-53.396,-178.531,6.253,148.696
C03202=1184.986,132.101,-53.417,-178.528,6.254,148.696
C03203=1184.980,132.370,-53.438,-178.526,6.256,148.696
C03204=1184.976,132.638,-53.460,-178.523,6.257,148.695
C03205=1184.970,132.907,-53.482,-178.520,6.259,148.695
C03206=1184.965,133.175,-53.503,-178.517,6.261,148.694
C03207=1184.961,133.424,-53.523,-178.514,6.262,148.694
C03208=1184.956,133.673,-53.544,-178.511,6.264,148.693
C03209=1184.950,133.922,-53.564,-178.509,6.265,148.693
C03210=1184.946,134.171,-53.584,-178.506,6.267,148.692
C03211=1184.941,134.421,-53.604,-178.503,6.268,148.692
C03212=1184.936,134.670,-53.624,-178.501,6.270,148.691
C03213=1184.932,134.919,-53.644,-178.498,6.271,148.691
C03214=1184.927,135.169,-53.665,-178.496,6.273,148.691
C03215=1184.922,135.418,-53.685,-178.493,6.274,148.690
C03216=1184.918,135.667,-53.705,-178.490,6.276,148.690
C03217=1184.913,135.916,-53.726,-178.488,6.277,148.689
C03218=1184.907,136.165,-53.746,-178.485,6.279,148.689
C03219=1184.903,136.414,-53.766,-178.482,6.280,148.689
C03220=1184.898,136.663,-53.786,-178.479,6.282,148.688
C03221=1184.894,136.912,-53.807,-178.477,6.283,148.687
C03222=1184.888,137.161,-53.827,-178.474,6.284,148.687
C03223=1184.884,137.410,-53.847,-178.472,6.286,148.687
C03224=1184.879,137.659,-53.868,-178.469,6.288,148.686
C03225=1184.874,137.909,-53.889,-178.466,6.289,148.686
C03226=1184.870,138.158,-53.908,-178.464,6.290,148.685
C03227=1184.865,138.407,-53.929,-178.461,6.292,148.685
C03228=1184.861,138.656,-53.949,-178.458,6.294,148.685
C03229=1184.856,138.905,-53.970,-178.456,6.295,148.684
C03230=1184.851,139.154,-53.990,-178.453,6.296,148.684
C03231=1184.847,139.403,-54.011,-178.450,6.298,148.683
C03232=1184.841,139.653,-54.032,-178.448,6.300,148.683
C03233=1184.837,139.902,-54.051,-178.445,6.301,148.682
C03234=1184.832,140.151,-54.072,-178.443,6.302,148.682
C03235=1184.827,140.400,-54.093,-178.440,6.304,148.681
C03236=1184.823,140.649,-54.113,-178.437,6.306,148.681
C03237=1184.818,140.899,-54.134,-178.434,6.307,148.681
C03238=1184.813,141.147,-54.155,-178.432,6.308,148.680
C03239=1184.809,141.396,-54.175,-178.429,6.310,148.680
C03240=1184.803,141.646,-54.196,-178.426,6.311,148.679
C03241=1184.799,141.895,-54.216,-178.424,6.313,148.679
C03242=1184.794,142.144,-54.237,-178.421,6.315,148.678
C03243=1184.789,142.393,-54.258,-178.419,6.316,148.678
C03244=1184.785,142.642,-54.278,-178.416,6.318,148.678
C03245=1184.780,142.891,-54.299,-178.413,6.319,148.677
C03246=1184.775,143.140,-54.319,-178.410,6.321,148.677
C03247=1184.770,143.389,-54.340,-178.408,6.323,148.676
C03248=1184.766,143.638,-54.361,-178.405,6.323,148.676
C03249=1184.761,143.887,-54.382,-178.403,6.325,148.675
C03250=1184.756,144.136,-54.402,-178.400,6.327,148.675
C03251=1184.751,144.386,-54.423,-178.397,6.328,148.674
C03252=1184.747,144.635,-54.443,-178.394,6.330,148.674
C03253=1184.742,144.884,-54.464,-178.392,6.331,148.674
C03254=1184.737,145.133,-54.485,-178.389,6.333,148.673
C03255=1184.732,145.382,-54.505,-178.387,6.335,148.673
C03256=1184.728,145.630,-54.527,-178.384,6.336,148.673
C03257=1184.723,145.879,-54.547,-178.381,6.338,148.672
C03258=1184.719,146.129,-54.568,-178.378,6.340,148.672
C03259=1184.713,146.379,-54.589,-178.376,6.341,148.671
C03260=1184.709,146.628,-54.610,-178.373,6.342,148.671
C03261=1184.704,146.877,-54.631,-178.371,6.344,148.670
C03262=1184.699,147.126,-54.651,-178.368,6.346,148.670
C03263=1184.695,147.374,-54.673,-178.365,6.348,148.670
C03264=1184.690,147.623,-54.693,-178.362,6.349,148.669
C03265=1184.685,147.873,-54.714,-178.360,6.350,148.669
C03266=1184.680,148.122,-54.735,-178.357,6.352,148.668
C03267=1184.676,148.371,-54.757,-178.355,6.353,148.668
C03268=1184.671,148.620,-54.777,-178.352,6.355,148.668
C03269=1184.667,148.869,-54.798,-178.349,6.357,148.667
C03270=1184.661,149.118,-54.819,-178.347,6.359,148.667
C03271=1184.657,149.367,-54.841,-178.344,6.359,148.666
C03272=1184.652,149.616,-54.861,-178.341,6.361,148.666
C03273=1184.647,149.865,-54.882,-178.339,6.363,148.665
C03274=1184.643,150.114,-54.903,-178.336,6.365,148.665
C03275=1184.638,150.363,-54.924,-178.333,6.366,148.665
C03276=1184.633,150.613,-54.945,-178.331,6.368,148.664
C03277=1184.629,150.861,-54.966,-178.328,6.369,148.664
C03278=1184.624,151.110,-54.987,-178.326,6.371,148.663
C03279=1184.619,151.360,-55.008,-178.323,6.372,148.663
C03280=1184.614,151.609,-55.030,-178.320,6.374,148.662
C03281=1184.610,151.858,-55.051,-178.317,6.376,148.662
C03282=1184.605,152.107,-55.072,-178.314,6.378,148.662
C03283=1184.600,152.356,-55.093,-178.312,6.379,148.661
C03284=1184.595,152.605,-55.114,-178.310,6.380,148.661
C03285=1184.591,152.854,-55.136,-178.307,6.382,148.661
C03286=1184.586,153.103,-55.157,-178.304,6.384,148.660
C03287=1184.581,153.352,-55.178,-178.301,6.385,148.660
C03288=1184.577,153.601,-55.199,-178.298,6.387,148.659
C03289=1184.571,153.850,-55.220,-178.296,6.389,148.659
C03290=1184.567,154.100,-55.242,-178.293,6.391,148.658
C03291=1184.562,154.349,-55.263,-178.290,6.392,148.658
C03292=1184.558,154.597,-55.284,-178.288,6.393,148.658
C03293=1184.553,154.846,-55.305,-178.286,6.395,148.657
C03294=1184.548,155.096,-55.327,-178.283,6.397,148.657
C03295=1184.544,155.344,-55.349,-178.280,6.399,148.657
C03296=1184.538,155.594,-55.369,-178.278,6.400,148.656
C03297=1184.534,155.842,-55.391,-178.274,6.402,148.656
C03298=1184.530,156.092,-55.412,-178.272,6.404,148.655
C03299=1184.525,156.341,-55.434,-178.269,6.405,148.655
C03300=1184.520,156.590,-55.455,-178.266,6.407,148.654
C03301=1184.515,156.839,-55.477,-178.264,6.408,148.654
C03302=1184.511,157.088,-55.498,-178.262,6.410,148.654
C03303=1184.506,157.337,-55.519,-178.259,6.412,148.653
C03304=1184.501,157.585,-55.540,-178.256,6.413,148.653
C03305=1184.497,157.835,-55.562,-178.253,6.415,148.653
C03306=1184.492,158.084,-55.583,-178.251,6.417,148.652
C03307=1184.487,158.353,-55.606,-178.248,6.418,148.652
C03308=1184.482,158.622,-55.630,-178.245,6.420,148.651
C03309=1184.477,158.891,-55.653,-178.242,6.422,148.651
C03310=1184.472,159.160,-55.676,-178.240,6.424,148.651
C03311=1184.467,159.409,-55.698,-178.237,6.425,148.650
C03312=1184.462,159.657,-55.720,-178.234,6.427,148.650
C03313=1184.457,159.907,-55.741,-178.232,6.429,148.649
C03314=1184.452,160.156,-55.763,-178.228,6.430,148.649
C03315=1184.448,160.405,-55.785,-178.226,6.432,148.648
C03316=1184.443,160.654,-55.806,-178.223,6.434,148.648
C03317=1184.438,160.903,-55.827,-178.220,6.436,148.648
C03318=1184.434,161.153,-55.849,-178.218,6.437,148.647
C03319=1184.430,161.401,-55.871,-178.215,6.439,148.647
C03320=1184.425,161.650,-55.892,-178.212,6.441,148.647
C03321=1184.421,161.899,-55.914,-178.210,6.443,148.646
C03322=1184.416,162.148,-55.936,-178.207,6.444,148.646
C03323=1184.411,162.398,-55.957,-178.205,6.446,148.645
C03324=1184.406,162.646,-55.979,-178.202,6.447,148.645
C03325=1184.401,162.895,-56.001,-178.199,6.449,148.645
C03326=1184.397,163.144,-56.023,-178.197,6.451,148.644
C03327=1184.392,163.393,-56.045,-178.194,6.453,148.644
C03328=1184.387,163.642,-56.067,-178.191,6.454,148.644
C03329=1184.382,163.891,-56.089,-178.189,6.456,148.643
C03330=1184.378,164.140,-56.110,-178.186,6.458,148.643
C03331=1184.373,164.389,-56.132,-178.183,6.460,148.642
C03332=1184.368,164.638,-56.153,-178.181,6.461,148.642
C03333=1184.364,164.888,-56.175,-178.178,6.463,148.642
C03334=1184.359,165.136,-56.197,-178.175,6.465,148.641
C03335=1184.355,165.386,-56.219,-178.173,6.467,148.641
C03336=1184.350,165.634,-56.241,-178.169,6.468,148.640
C03337=1184.346,165.884,-56.263,-178.167,6.470,148.640
C03338=1184.341,166.132,-56.285,-178.164,6.472,148.640
C03339=1184.336,166.381,-56.306,-178.161,6.474,148.639
C03340=1184.331,166.631,-56.329,-178.159,6.475,148.639
C03341=1184.326,166.879,-56.351,-178.157,6.476,148.639
C03342=1184.322,167.129,-56.373,-178.154,6.478,148.638
C03343=1184.317,167.377,-56.395,-178.151,6.480,148.638
C03344=1184.313,167.626,-56.417,-178.149,6.482,148.637
C03345=1184.308,167.875,-56.439,-178.146,6.483,148.637
C03346=1184.304,168.124,-56.461,-178.143,6.485,148.637
C03347=1184.298,168.373,-56.483,-178.141,6.487,148.636
C03348=1184.294,168.622,-56.505,-178.138,6.489,148.636
C03349=1184.289,168.871,-56.527,-178.135,6.490,148.636
C03350=1184.285,169.120,-56.549,-178.133,6.492,148.635
C03351=1184.280,169.369,-56.571,-178.130,6.494,148.635
C03352=1184.275,169.618,-56.594,-178.127,6.496,148.635
C03353=1184.270,169.866,-56.616,-178.125,6.498,148.634
C03354=1184.266,170.116,-56.638,-178.122,6.499,148.634
C03355=1184.261,170.364,-56.659,-178.119,6.501,148.633
C03356=1184.256,170.614,-56.682,-178.116,6.503,148.633
C03357=1184.252,170.863,-56.705,-178.114,6.505,148.633
C03358=1184.247,171.111,-56.726,-178.111,6.506,148.632
C03359=1184.243,171.361,-56.748,-178.108,6.508,148.632
C03360=1184.237,171.610,-56.771,-178.106,6.510,148.632
C03361=1184.233,171.858,-56.794,-178.103,6.512,148.631
C03362=1184.229,172.107,-56.815,-178.100,6.514,148.631
C03363=1184.224,172.357,-56.838,-178.098,6.515,148.630
C03364=1184.219,172.606,-56.860,-178.095,6.517,148.630
C03365=1184.215,172.854,-56.882,-178.092,6.519,148.630
C03366=1184.210,173.104,-56.905,-178.090,6.521,148.629
C03367=1184.205,173.352,-56.927,-178.088,6.523,148.629
C03368=1184.201,173.601,-56.949,-178.085,6.525,148.629
C03369=1184.196,173.851,-56.972,-178.082,6.526,148.629
C03370=1184.191,174.099,-56.994,-178.079,6.528,148.628
C03371=1184.187,174.348,-57.016,-178.077,6.530,148.628
C03372=1184.181,174.597,-57.039,-178.074,6.532,148.627
C03373=1184.177,174.846,-57.061,-178.071,6.534,148.627
C03374=1184.173,175.095,-57.084,-178.069,6.535,148.627
C03375=1184.168,175.344,-57.106,-178.066,6.537,148.626
C03376=1184.164,175.593,-57.129,-178.063,6.539,148.626
C03377=1184.159,175.843,-57.151,-178.061,6.541,148.626
C03378=1184.154,176.091,-57.174,-178.058,6.542,148.625
C03379=1184.150,176.340,-57.196,-178.055,6.544,148.625
C03380=1184.144,176.588,-57.219,-178.053,6.546,148.625
C03381=1184.140,176.838,-57.241,-178.050,6.548,148.624
C03382=1184.136,177.087,-57.264,-178.047,6.550,148.624
C03383=1184.131,177.335,-57.286,-178.045,6.551,148.623
C03384=1184.126,177.584,-57.309,-178.042,6.553,148.623
C03385=1184.122,177.834,-57.331,-178.039,6.555,148.623
C03386=1184.117,178.083,-57.355,-178.036,6.558,148.622
C03387=1184.112,178.331,-57.376,-178.033,6.559,148.622
C03388=1184.107,178.580,-57.400,-178.031,6.561,148.622
C03389=1184.103,178.830,-57.422,-178.029,6.563,148.622
C03390=1184.098,179.078,-57.445,-178.026,6.565,148.621
C03391=1184.094,179.327,-57.467,-178.023,6.567,148.621
C03392=1184.089,179.576,-57.490,-178.021,6.569,148.620
C03393=1184.084,179.824,-57.512,-178.018,6.570,148.620
C03394=1184.079,180.074,-57.535,-178.015,6.572,148.620
C03395=1184.075,180.323,-57.558,-178.013,6.574,148.619
C03396=1184.071,180.572,-57.581,-178.010,6.576,148.619
C03397=1184.066,180.820,-57.603,-178.007,6.577,148.619
C03398=1184.061,181.069,-57.626,-178.005,6.579,148.618
C03399=1184.057,181.318,-57.649,-178.002,6.581,148.618
C03400=1184.052,181.568,-57.672,-177.999,6.583,148.618
C03401=1184.048,181.816,-57.694,-177.997,6.585,148.617
C03402=1184.043,182.065,-57.717,-177.994,6.587,148.617
C03403=1184.038,182.315,-57.740,-177.992,6.589,148.617
C03404=1184.034,182.563,-57.763,-177.988,6.591,148.616
C03405=1184.029,182.812,-57.786,-177.986,6.593,148.616
C03406=1184.025,183.060,-57.809,-177.983,6.595,148.616
C03407=1184.020,183.310,-57.831,-177.980,6.596,148.615
C03408=1184.015,183.559,-57.855,-177.978,6.598,148.615
C03409=1184.011,183.808,-57.877,-177.975,6.600,148.615
C03410=1184.006,184.056,-57.900,-177.972,6.602,148.614
C03411=1184.000,184.326,-57.925,-177.970,6.604,148.614
C03412=1183.996,184.595,-57.950,-177.966,6.606,148.614
C03413=1183.990,184.865,-57.975,-177.964,6.608,148.613
C03414=1183.986,185.135,-58.000,-177.961,6.610,148.613
C03415=1183.981,185.383,-58.023,-177.958,6.612,148.613
C03416=1183.976,185.633,-58.046,-177.955,6.614,148.612
C03417=1183.972,185.882,-58.069,-177.953,6.616,148.612
C03418=1183.968,186.130,-58.092,-177.950,6.618,148.612
C03419=1183.963,186.379,-58.115,-177.948,6.620,148.611
C03420=1183.958,186.628,-58.139,-177.945,6.622,148.611
C03421=1183.953,186.877,-58.162,-177.942,6.623,148.611
C03422=1183.949,187.125,-58.185,-177.940,6.625,148.610
C03423=1183.944,187.375,-58.207,-177.937,6.627,148.610
C03424=1183.939,187.624,-58.231,-177.934,6.629,148.610
C03425=1183.935,187.873,-58.254,-177.932,6.631,148.609
C03426=1183.931,188.122,-58.277,-177.929,6.634,148.609
C03427=1183.926,188.371,-58.300,-177.926,6.635,148.609
C03428=1183.921,188.619,-58.323,-177.924,6.637,148.608
C03429=1183.916,188.868,-58.346,-177.921,6.639,148.608
C03430=1183.911,189.117,-58.370,-177.918,6.641,148.608
C03431=1183.908,189.365,-58.393,-177.916,6.643,148.607
C03432=1183.903,189.614,-58.417,-177.913,6.644,148.607
C03433=1183.898,189.863,-58.440,-177.911,6.646,148.607
C03434=1183.894,190.112,-58.463,-177.908,6.648,148.606
C03435=1183.889,190.361,-58.487,-177.905,6.651,148.606
C03436=1183.884,190.611,-58.510,-177.902,6.653,148.606
C03437=1183.880,190.859,-58.533,-177.899,6.654,148.605
C03438=1183.876,191.108,-58.556,-177.897,6.656,148.605
C03439=1183.870,191.357,-58.579,-177.894,6.658,148.605
C03440=1183.866,191.606,-58.603,-177.892,6.660,148.605
C03441=1183.861,191.854,-58.627,-177.889,6.662,148.604
C03442=1183.856,192.103,-58.650,-177.887,6.664,148.604
C03443=1183.852,192.352,-58.673,-177.883,6.666,148.604
C03444=1183.847,192.601,-58.697,-177.881,6.668,148.603
C03445=1183.842,192.850,-58.720,-177.878,6.670,148.603
C03446=1183.838,193.099,-58.744,-177.876,6.672,148.603
C03447=1183.834,193.347,-58.767,-177.873,6.674,148.602
C03448=1183.829,193.596,-58.790,-177.871,6.676,148.602
C03449=1183.825,193.845,-58.814,-177.868,6.677,148.602
C03450=1183.820,194.094,-58.838,-177.865,6.680,148.601
C03451=1183.815,194.343,-58.861,-177.862,6.682,148.601
C03452=1183.811,194.592,-58.884,-177.860,6.684,148.601
C03453=1183.806,194.841,-58.908,-177.857,6.686,148.601
C03454=1183.802,195.089,-58.932,-177.854,6.688,148.600
C03455=1183.797,195.338,-58.955,-177.852,6.689,148.600
C03456=1183.792,195.587,-58.979,-177.849,6.692,148.600
C03457=1183.788,195.836,-59.003,-177.846,6.694,148.599
C03458=1183.783,196.085,-59.026,-177.844,6.696,148.599
C03459=1183.779,196.334,-59.049,-177.841,6.698,148.599
C03460=1183.774,196.582,-59.073,-177.838,6.700,148.598
C03461=1183.769,196.831,-59.097,-177.836,6.701,148.598
C03462=1183.765,197.080,-59.121,-177.833,6.704,148.598
C03463=1183.760,197.329,-59.144,-177.830,6.706,148.598
C03464=1183.755,197.578,-59.168,-177.828,6.708,148.597
C03465=1183.751,197.827,-59.193,-177.825,6.710,148.597
C03466=1183.746,198.076,-59.216,-177.822,6.711,148.597
C03467=1183.742,198.325,-59.240,-177.820,6.714,148.596
C03468=1183.737,198.574,-59.263,-177.817,6.716,148.596
C03469=1183.733,198.822,-59.287,-177.814,6.718,148.596
C03470=1183.728,199.071,-59.311,-177.812,6.720,148.595
C03471=1183.724,199.320,-59.335,-177.809,6.722,148.595
C03472=1183.719,199.569,-59.358,-177.807,6.724,148.595
C03473=1183.715,199.817,-59.382,-177.803,6.726,148.595
C03474=1183.709,200.066,-59.406,-177.801,6.728,148.594
C03475=1183.705,200.315,-59.430,-177.798,6.730,148.594
C03476=1183.701,200.564,-59.454,-177.796,6.732,148.594
C03477=1183.696,200.813,-59.478,-177.793,6.734,148.593
C03478=1183.692,201.061,-59.502,-177.790,6.736,148.593
C03479=1183.687,201.310,-59.526,-177.787,6.738,148.593
C03480=1183.682,201.559,-59.550,-177.785,6.740,148.592
C03481=1183.677,201.808,-59.574,-177.783,6.742,148.592
C03482=1183.673,202.056,-59.598,-177.780,6.744,148.592
C03483=1183.669,202.306,-59.622,-177.777,6.747,148.592
C03484=1183.665,202.555,-59.645,-177.774,6.748,148.591
C03485=1183.659,202.803,-59.670,-177.772,6.751,148.591
C03486=1183.655,203.052,-59.694,-177.769,6.752,148.591
C03487=1183.650,203.301,-59.718,-177.766,6.754,148.590
C03488=1183.646,203.549,-59.742,-177.763,6.757,148.590
C03489=1183.641,203.799,-59.767,-177.761,6.759,148.590
C03490=1183.637,204.047,-59.791,-177.758,6.761,148.590
C03491=1183.632,204.296,-59.814,-177.756,6.762,148.589
C03492=1183.628,204.544,-59.838,-177.753,6.764,148.589
C03493=1183.623,204.793,-59.863,-177.750,6.767,148.589
C03494=1183.619,205.042,-59.887,-177.748,6.769,148.589
C03495=1183.614,205.291,-59.911,-177.745,6.771,148.588
C03496=1183.609,205.540,-59.935,-177.742,6.773,148.588
C03497=1183.605,205.788,-59.959,-177.740,6.776,148.588
C03498=1183.600,206.037,-59.983,-177.737,6.777,148.587
C03499=1183.596,206.286,-60.009,-177.734,6.779,148.587
C03500=1183.591,206.535,-60.032,-177.732,6.781,148.587
C03501=1183.587,206.784,-60.056,-177.729,6.784,148.587
C03502=1183.582,207.033,-60.081,-177.726,6.786,148.586
C03503=1183.578,207.282,-60.105,-177.724,6.788,148.586
C03504=1183.573,207.530,-60.129,-177.721,6.790,148.586
C03505=1183.568,207.779,-60.154,-177.718,6.792,148.586
C03506=1183.564,208.027,-60.178,-177.715,6.794,148.585
C03507=1183.559,208.277,-60.203,-177.713,6.796,148.585
C03508=1183.555,208.525,-60.227,-177.711,6.798,148.585
C03509=1183.550,208.774,-60.250,-177.707,6.801,148.584
C03510=1183.545,209.023,-60.275,-177.705,6.802,148.584
C03511=1183.541,209.272,-60.299,-177.703,6.805,148.584
C03512=1183.536,209.521,-60.324,-177.700,6.806,148.584
C03513=1183.532,209.769,-60.348,-177.697,6.809,148.583
C03514=1183.527,210.018,-60.373,-177.694,6.811,148.583
C03515=1183.522,210.289,-60.400,-177.692,6.813,148.583
C03516=1183.518,210.558,-60.426,-177.689,6.816,148.583
C03517=1183.513,210.829,-60.453,-177.686,6.817,148.582
C03518=1183.508,211.100,-60.480,-177.683,6.820,148.582
C03519=1183.503,211.348,-60.505,-177.680,6.822,148.582
C03520=1183.499,211.597,-60.529,-177.677,6.825,148.581
C03521=1183.494,211.846,-60.554,-177.675,6.827,148.581
C03522=1183.490,212.094,-60.578,-177.672,6.828,148.581
C03523=1183.484,212.343,-60.602,-177.670,6.831,148.581
C03524=1183.481,212.592,-60.627,-177.667,6.833,148.580
C03525=1183.476,212.841,-60.651,-177.664,6.835,148.580
C03526=1183.471,213.089,-60.676,-177.661,6.837,148.580
C03527=1183.467,213.338,-60.701,-177.658,6.840,148.580
C03528=1183.463,213.587,-60.725,-177.656,6.842,148.579
C03529=1183.457,213.835,-60.750,-177.653,6.843,148.579
C03530=1183.453,214.085,-60.775,-177.651,6.845,148.579
C03531=1183.448,214.333,-60.799,-177.648,6.848,148.579
C03532=1183.444,214.582,-60.825,-177.645,6.850,148.578
C03533=1183.440,214.830,-60.849,-177.643,6.852,148.578
C03534=1183.435,215.079,-60.874,-177.640,6.855,148.578
C03535=1183.430,215.329,-60.899,-177.637,6.857,148.577
C03536=1183.426,215.576,-60.923,-177.635,6.859,148.577
C03537=1183.422,215.826,-60.949,-177.632,6.860,148.577
C03538=1183.416,216.075,-60.973,-177.629,6.863,148.577
C03539=1183.412,216.322,-60.998,-177.627,6.865,148.577
C03540=1183.408,216.572,-61.023,-177.624,6.867,148.576
C03541=1183.403,216.820,-61.047,-177.621,6.870,148.576
C03542=1183.399,217.069,-61.073,-177.619,6.872,148.576
C03543=1183.394,217.318,-61.098,-177.616,6.874,148.575
C03544=1183.390,217.567,-61.123,-177.613,6.877,148.575
C03545=1183.385,217.815,-61.147,-177.611,6.878,148.575
C03546=1183.381,218.064,-61.172,-177.608,6.880,148.575
C03547=1183.376,218.313,-61.197,-177.605,6.883,148.575
C03548=1183.372,218.562,-61.222,-177.603,6.885,148.574
C03549=1183.367,218.810,-61.247,-177.600,6.887,148.574
C03550=1183.362,219.058,-61.272,-177.598,6.889,148.574
C03551=1183.358,219.308,-61.297,-177.595,6.892,148.574
C03552=1183.354,219.556,-61.322,-177.592,6.893,148.573
C03553=1183.349,219.805,-61.347,-177.590,6.895,148.573
C03554=1183.344,220.053,-61.373,-177.587,6.898,148.573
C03555=1183.340,220.303,-61.398,-177.584,6.900,148.573
C03556=1183.336,220.550,-61.422,-177.582,6.902,148.572
C03557=1183.331,220.800,-61.447,-177.578,6.905,148.572
C03558=1183.327,221.049,-61.473,-177.576,6.907,148.572
C03559=1183.322,221.297,-61.498,-177.574,6.909,148.572
C03560=1183.318,221.546,-61.524,-177.570,6.911,148.571
C03561=1183.313,221.795,-61.548,-177.568,6.913,148.571
C03562=1183.309,222.043,-61.573,-177.566,6.915,148.571
C03563=1183.304,222.292,-61.598,-177.563,6.918,148.571
C03564=1183.300,222.541,-61.624,-177.560,6.920,148.570
C03565=1183.295,222.789,-61.649,-177.558,6.922,148.570
C03566=1183.290,223.038,-61.674,-177.555,6.925,148.570
C03567=1183.286,223.286,-61.699,-177.552,6.927,148.570
C03568=1183.282,223.536,-61.724,-177.549,6.930,148.570
C03569=1183.277,223.784,-61.749,-177.547,6.931,148.569
C03570=1183.273,224.032,-61.775,-177.545,6.934,148.569
C03571=1183.268,224.281,-61.801,-177.541,6.936,148.569
C03572=1183.263,224.530,-61.826,-177.539,6.938,148.569
C03573=1183.259,224.779,-61.851,-177.537,6.940,148.568
C03574=1183.254,225.027,-61.877,-177.533,6.943,148.568
C03575=1183.250,225.276,-61.902,-177.531,6.945,148.568
C03576=1183.245,225.525,-61.928,-177.528,6.947,148.568
C03577=1183.241,225.773,-61.953,-177.525,6.949,148.567
C03578=1183.236,226.022,-61.979,-177.523,6.951,148.567
C03579=1183.231,226.271,-62.003,-177.520,6.953,148.567
C03580=1183.227,226.520,-62.029,-177.518,6.956,148.567
C03581=1183.223,226.768,-62.055,-177.515,6.958,148.567
C03582=1183.219,227.016,-62.080,-177.512,6.961,148.566
C03583=1183.215,227.265,-62.105,-177.510,6.963,148.566
C03584=1183.210,227.514,-62.130,-177.507,6.965,148.566
C03585=1183.204,227.763,-62.156,-177.504,6.968,148.566
C03586=1183.200,228.012,-62.182,-177.502,6.969,148.565
C03587=1183.196,228.260,-62.208,-177.499,6.972,148.565
C03588=1183.191,228.509,-62.233,-177.496,6.974,148.565
C03589=1183.187,228.757,-62.259,-177.494,6.976,148.565
C03590=1183.183,229.006,-62.285,-177.491,6.979,148.565
C03591=1183.178,229.254,-62.310,-177.489,6.981,148.564
C03592=1183.174,229.503,-62.336,-177.486,6.983,148.564
C03593=1183.169,229.752,-62.362,-177.483,6.986,148.564
C03594=1183.164,230.001,-62.386,-177.481,6.988,148.564
C03595=1183.160,230.249,-62.412,-177.478,6.991,148.564
C03596=1183.156,230.498,-62.438,-177.475,6.993,148.563
C03597=1183.151,230.746,-62.463,-177.473,6.995,148.563
C03598=1183.147,230.995,-62.489,-177.470,6.997,148.563
C03599=1183.142,231.244,-62.515,-177.468,6.999,148.563
C03600=1183.138,231.493,-62.541,-177.464,7.002,148.563
C03601=1183.133,231.741,-62.567,-177.462,7.004,148.562
C03602=1183.129,231.989,-62.593,-177.460,7.006,148.562
C03603=1183.125,232.238,-62.619,-177.456,7.009,148.562
C03604=1183.120,232.486,-62.644,-177.454,7.011,148.562
C03605=1183.116,232.735,-62.670,-177.451,7.013,148.561
C03606=1183.111,232.984,-62.696,-177.449,7.016,148.561
C03607=1183.106,233.233,-62.722,-177.447,7.018,148.561
C03608=1183.102,233.481,-62.747,-177.443,7.020,148.561
C03609=1183.097,233.730,-62.773,-177.441,7.023,148.561
C03610=1183.093,233.979,-62.799,-177.438,7.025,148.561
C03611=1183.088,234.227,-62.826,-177.436,7.027,148.560
C03612=1183.084,234.476,-62.852,-177.433,7.030,148.560
C03613=1183.079,234.724,-62.877,-177.430,7.032,148.560
C03614=1183.075,234.973,-62.903,-177.428,7.034,148.560
C03615=1183.070,235.222,-62.929,-177.425,7.037,148.560
C03616=1183.066,235.470,-62.956,-177.422,7.039,148.559
C03617=1183.062,235.719,-62.981,-177.420,7.042,148.559
C03618=1183.057,235.967,-63.007,-177.417,7.044,148.559
C03619=1183.052,236.239,-63.036,-177.414,7.046,148.559
C03620=1183.047,236.511,-63.064,-177.411,7.049,148.559
C03621=1183.043,236.782,-63.092,-177.408,7.051,148.558
C03622=1183.038,237.054,-63.121,-177.406,7.054,148.558
C03623=1183.033,237.302,-63.147,-177.402,7.057,148.558
C03624=1183.029,237.550,-63.173,-177.400,7.059,148.558
C03625=1183.025,237.799,-63.199,-177.398,7.061,148.557
C03626=1183.020,238.048,-63.225,-177.395,7.063,148.557
C03627=1183.016,238.296,-63.252,-177.393,7.066,148.557
C03628=1183.011,238.546,-63.278,-177.390,7.068,148.557
C03629=1183.006,238.794,-63.304,-177.387,7.070,148.557
C03630=1183.002,239.042,-63.330,-177.384,7.073,148.557
C03631=1182.997,239.291,-63.356,-177.382,7.075,148.557
C03632=1182.993,239.539,-63.383,-177.379,7.078,148.556
C03633=1182.989,239.788,-63.409,-177.377,7.080,148.556
C03634=1182.984,240.037,-63.435,-177.374,7.083,148.556
C03635=1182.980,240.285,-63.461,-177.371,7.085,148.556
C03636=1182.975,240.534,-63.488,-177.369,7.087,148.556
C03637=1182.971,240.783,-63.514,-177.366,7.090,148.555
C03638=1182.966,241.031,-63.540,-177.364,7.092,148.555
C03639=1182.962,241.279,-63.567,-177.361,7.095,148.555
C03640=1182.958,241.528,-63.592,-177.358,7.097,148.555
C03641=1182.953,241.776,-63.620,-177.356,7.100,148.555
C03642=1182.949,242.025,-63.645,-177.353,7.101,148.554
C03643=1182.944,242.274,-63.672,-177.350,7.104,148.554
C03644=1182.940,242.522,-63.699,-177.347,7.106,148.554
C03645=1182.935,242.771,-63.725,-177.345,7.109,148.554
C03646=1182.931,243.019,-63.752,-177.343,7.111,148.554
C03647=1182.926,243.268,-63.778,-177.339,7.114,148.554
C03648=1182.922,243.517,-63.804,-177.337,7.116,148.554
C03649=1182.918,243.765,-63.831,-177.334,7.119,148.553
C03650=1182.913,244.014,-63.857,-177.332,7.121,148.553
C03651=1182.909,244.262,-63.884,-177.329,7.124,148.553
C03652=1182.904,244.511,-63.911,-177.326,7.126,148.553
C03653=1182.900,244.760,-63.937,-177.324,7.129,148.553
C03654=1182.895,245.008,-63.964,-177.322,7.131,148.553
C03655=1182.891,245.256,-63.991,-177.318,7.133,148.552
C03656=1182.886,245.505,-64.017,-177.316,7.136,148.552
C03657=1182.882,245.754,-64.043,-177.313,7.139,148.552
